Yaskawa INFORM job: A_ROOF_UPPER_0614_2_PAINT_29.JBI

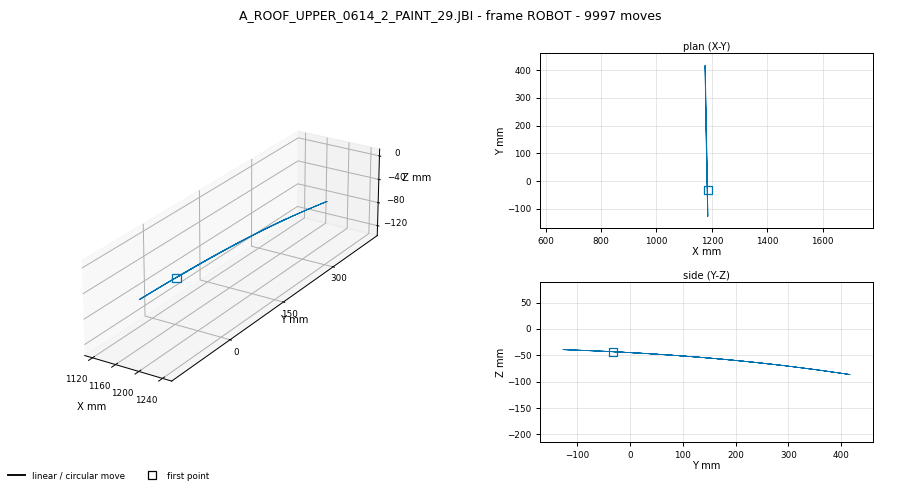
[picture p0: tool path of A_ROOF_UPPER_0614_2_PAINT_29.JBI in frame ROBOT, 9997 of 9997 moves have a stored position in this frame; points joined in program order, loops and branches not executed]
/JOB
//NAME A_ROOF_UPPER_0614_2_PAINT29
//POS
///NPOS 9997,0,0,0,0,0
///TOOL 1
///USER 0
///POSTYPE ROBOT
///RECTAN
///RCONF 1,0,0,0,0,0,0,0,0,0,0,0,0,0,0,0,0,0,0,0,0,0,0,0
C00000=1184.882,-32.072,-43.136,179.748,5.725,149.090
C00001=1184.877,-31.822,-43.149,179.750,5.725,149.089
C00002=1184.871,-31.573,-43.161,179.753,5.726,149.088
C00003=1184.866,-31.323,-43.173,179.755,5.726,149.088
C00004=1184.861,-31.074,-43.186,179.758,5.727,149.087
C00005=1184.855,-30.824,-43.198,179.760,5.727,149.086
C00006=1184.850,-30.574,-43.210,179.762,5.727,149.086
C00007=1184.846,-30.324,-43.223,179.765,5.728,149.085
C00008=1184.840,-30.074,-43.235,179.767,5.728,149.084
C00009=1184.835,-29.825,-43.248,179.770,5.729,149.084
C00010=1184.830,-29.576,-43.260,179.772,5.729,149.083
C00011=1184.825,-29.326,-43.272,179.775,5.730,149.083
C00012=1184.820,-29.077,-43.285,179.777,5.730,149.082
C00013=1184.815,-28.827,-43.298,179.780,5.730,149.081
C00014=1184.810,-28.577,-43.311,179.782,5.731,149.081
C00015=1184.804,-28.327,-43.322,179.784,5.731,149.080
C00016=1184.799,-28.078,-43.335,179.787,5.732,149.079
C00017=1184.794,-27.829,-43.348,179.789,5.733,149.079
C00018=1184.789,-27.579,-43.360,179.791,5.732,149.078
C00019=1184.784,-27.329,-43.372,179.794,5.733,149.077
C00020=1184.779,-27.079,-43.385,179.797,5.733,149.077
C00021=1184.773,-26.830,-43.398,179.799,5.734,149.076
C00022=1184.768,-26.580,-43.411,179.801,5.734,149.076
C00023=1184.763,-26.331,-43.423,179.804,5.735,149.075
C00024=1184.758,-26.081,-43.436,179.806,5.735,149.074
C00025=1184.753,-25.831,-43.448,179.808,5.735,149.074
C00026=1184.748,-25.582,-43.461,179.811,5.736,149.073
C00027=1184.743,-25.333,-43.474,179.814,5.736,149.072
C00028=1184.738,-25.083,-43.486,179.816,5.737,149.072
C00029=1184.732,-24.832,-43.499,179.819,5.738,149.071
C00030=1184.727,-24.583,-43.512,179.821,5.737,149.070
C00031=1184.722,-24.334,-43.524,179.823,5.738,149.070
C00032=1184.717,-24.084,-43.537,179.825,5.738,149.069
C00033=1184.712,-23.815,-43.550,179.828,5.739,149.069
C00034=1184.706,-23.545,-43.565,179.831,5.739,149.068
C00035=1184.701,-23.275,-43.578,179.833,5.740,149.067
C00036=1184.694,-23.005,-43.592,179.836,5.740,149.066
C00037=1184.689,-22.756,-43.604,179.839,5.741,149.066
C00038=1184.685,-22.506,-43.617,179.841,5.741,149.065
C00039=1184.680,-22.256,-43.630,179.844,5.742,149.065
C00040=1184.674,-22.007,-43.642,179.846,5.742,149.064
C00041=1184.669,-21.757,-43.656,179.848,5.742,149.063
C00042=1184.664,-21.507,-43.669,179.851,5.743,149.063
C00043=1184.659,-21.258,-43.681,179.853,5.743,149.062
C00044=1184.654,-21.009,-43.694,179.856,5.744,149.061
C00045=1184.649,-20.758,-43.707,179.858,5.744,149.061
C00046=1184.643,-20.509,-43.720,179.861,5.745,149.060
C00047=1184.638,-20.260,-43.732,179.863,5.745,149.060
C00048=1184.634,-20.010,-43.745,179.865,5.745,149.059
C00049=1184.628,-19.760,-43.759,179.868,5.746,149.058
C00050=1184.623,-19.511,-43.771,179.870,5.747,149.058
C00051=1184.618,-19.261,-43.784,179.873,5.747,149.057
C00052=1184.612,-19.011,-43.797,179.876,5.747,149.056
C00053=1184.607,-18.762,-43.810,179.878,5.748,149.056
C00054=1184.602,-18.512,-43.823,179.880,5.749,149.055
C00055=1184.598,-18.262,-43.836,179.882,5.748,149.054
C00056=1184.592,-18.013,-43.849,179.885,5.749,149.054
C00057=1184.587,-17.763,-43.861,179.887,5.750,149.053
C00058=1184.582,-17.513,-43.874,179.890,5.750,149.053
C00059=1184.576,-17.264,-43.888,179.893,5.751,149.052
C00060=1184.571,-17.015,-43.900,179.895,5.751,149.051
C00061=1184.567,-16.764,-43.913,179.897,5.752,149.051
C00062=1184.561,-16.515,-43.926,179.900,5.752,149.050
C00063=1184.556,-16.266,-43.940,179.902,5.752,149.049
C00064=1184.551,-16.016,-43.953,179.905,5.753,149.049
C00065=1184.546,-15.767,-43.966,179.907,5.753,149.048
C00066=1184.541,-15.516,-43.979,179.910,5.754,149.047
C00067=1184.536,-15.267,-43.991,179.912,5.754,149.047
C00068=1184.530,-15.018,-44.005,179.915,5.755,149.046
C00069=1184.526,-14.768,-44.018,179.917,5.756,149.046
C00070=1184.520,-14.518,-44.030,179.920,5.756,149.045
C00071=1184.515,-14.269,-44.044,179.922,5.757,149.044
C00072=1184.510,-14.019,-44.057,179.924,5.757,149.044
C00073=1184.505,-13.770,-44.070,179.927,5.757,149.043
C00074=1184.500,-13.520,-44.083,179.929,5.757,149.042
C00075=1184.495,-13.270,-44.096,179.932,5.758,149.042
C00076=1184.489,-13.021,-44.110,179.934,5.759,149.041
C00077=1184.485,-12.771,-44.123,179.937,5.759,149.041
C00078=1184.479,-12.522,-44.136,179.940,5.760,149.040
C00079=1184.474,-12.272,-44.149,179.942,5.761,149.039
C00080=1184.469,-12.023,-44.163,179.944,5.761,149.039
C00081=1184.464,-11.773,-44.176,179.947,5.761,149.038
C00082=1184.459,-11.523,-44.188,179.949,5.761,149.037
C00083=1184.453,-11.274,-44.201,179.951,5.762,149.037
C00084=1184.449,-11.024,-44.215,179.954,5.762,149.036
C00085=1184.443,-10.775,-44.228,179.957,5.763,149.035
C00086=1184.439,-10.525,-44.241,179.959,5.763,149.035
C00087=1184.433,-10.275,-44.255,179.961,5.764,149.034
C00088=1184.429,-10.025,-44.268,179.964,5.765,149.034
C00089=1184.423,-9.776,-44.281,179.967,5.765,149.033
C00090=1184.418,-9.526,-44.294,179.969,5.766,149.032
C00091=1184.413,-9.277,-44.308,179.972,5.766,149.032
C00092=1184.408,-9.027,-44.321,179.974,5.767,149.031
C00093=1184.402,-8.777,-44.334,179.976,5.767,149.030
C00094=1184.398,-8.528,-44.348,179.978,5.767,149.030
C00095=1184.392,-8.278,-44.361,179.981,5.768,149.029
C00096=1184.387,-8.029,-44.374,179.984,5.768,149.029
C00097=1184.382,-7.779,-44.388,179.986,5.769,149.028
C00098=1184.377,-7.530,-44.401,179.989,5.770,149.027
C00099=1184.372,-7.280,-44.415,179.991,5.770,149.027
C00100=1184.367,-7.031,-44.428,179.994,5.771,149.026
C00101=1184.362,-6.780,-44.441,179.996,5.771,149.026
C00102=1184.357,-6.532,-44.455,179.999,5.772,149.025
C00103=1184.352,-6.281,-44.468,-179.999,5.772,149.024
C00104=1184.346,-6.032,-44.482,-179.996,5.773,149.023
C00105=1184.342,-5.782,-44.495,-179.994,5.774,149.023
C00106=1184.337,-5.533,-44.509,-179.992,5.773,149.022
C00107=1184.331,-5.283,-44.522,-179.989,5.774,149.022
C00108=1184.327,-5.034,-44.536,-179.987,5.775,149.021
C00109=1184.321,-4.784,-44.549,-179.984,5.775,149.020
C00110=1184.316,-4.534,-44.562,-179.982,5.776,149.020
C00111=1184.311,-4.285,-44.576,-179.979,5.776,149.019
C00112=1184.306,-4.035,-44.589,-179.977,5.777,149.019
C00113=1184.301,-3.786,-44.603,-179.974,5.777,149.018
C00114=1184.295,-3.536,-44.617,-179.971,5.778,149.017
C00115=1184.290,-3.287,-44.630,-179.969,5.778,149.017
C00116=1184.285,-3.037,-44.644,-179.967,5.779,149.016
C00117=1184.280,-2.788,-44.657,-179.964,5.780,149.015
C00118=1184.275,-2.538,-44.671,-179.961,5.780,149.015
C00119=1184.270,-2.288,-44.685,-179.959,5.781,149.014
C00120=1184.265,-2.039,-44.698,-179.957,5.781,149.014
C00121=1184.260,-1.789,-44.712,-179.954,5.782,149.013
C00122=1184.255,-1.540,-44.725,-179.951,5.782,149.012
C00123=1184.250,-1.290,-44.738,-179.949,5.783,149.012
C00124=1184.245,-1.040,-44.753,-179.947,5.783,149.011
C00125=1184.239,-0.791,-44.767,-179.944,5.783,149.010
C00126=1184.234,-0.541,-44.780,-179.942,5.784,149.010
C00127=1184.229,-0.292,-44.794,-179.939,5.785,149.009
C00128=1184.224,-0.042,-44.808,-179.937,5.785,149.008
C00129=1184.219,0.208,-44.821,-179.934,5.786,149.008
C00130=1184.214,0.457,-44.835,-179.932,5.787,149.007
C00131=1184.209,0.707,-44.848,-179.929,5.787,149.007
C00132=1184.204,0.956,-44.862,-179.927,5.787,149.006
C00133=1184.199,1.206,-44.876,-179.925,5.788,149.006
C00134=1184.194,1.456,-44.889,-179.922,5.789,149.005
C00135=1184.189,1.705,-44.903,-179.919,5.789,149.004
C00136=1184.184,1.954,-44.918,-179.917,5.790,149.003
C00137=1184.178,2.224,-44.933,-179.914,5.790,149.003
C00138=1184.172,2.493,-44.947,-179.912,5.791,149.002
C00139=1184.167,2.762,-44.962,-179.909,5.792,149.002
C00140=1184.162,3.031,-44.977,-179.906,5.793,149.001
C00141=1184.157,3.281,-44.991,-179.903,5.793,149.000
C00142=1184.151,3.530,-45.005,-179.901,5.794,149.000
C00143=1184.146,3.780,-45.018,-179.898,5.795,148.999
C00144=1184.141,4.030,-45.033,-179.896,5.795,148.998
C00145=1184.136,4.279,-45.046,-179.894,5.795,148.998
C00146=1184.131,4.528,-45.060,-179.891,5.795,148.997
C00147=1184.126,4.779,-45.074,-179.889,5.796,148.997
C00148=1184.121,5.028,-45.088,-179.886,5.797,148.996
C00149=1184.116,5.277,-45.102,-179.884,5.797,148.995
C00150=1184.111,5.527,-45.116,-179.881,5.798,148.995
C00151=1184.106,5.776,-45.130,-179.879,5.798,148.994
C00152=1184.101,6.026,-45.143,-179.876,5.799,148.993
C00153=1184.096,6.276,-45.157,-179.873,5.799,148.993
C00154=1184.091,6.525,-45.172,-179.871,5.800,148.992
C00155=1184.085,6.774,-45.186,-179.869,5.801,148.992
C00156=1184.080,7.024,-45.200,-179.866,5.801,148.991
C00157=1184.075,7.274,-45.214,-179.864,5.802,148.990
C00158=1184.070,7.523,-45.227,-179.861,5.802,148.990
C00159=1184.065,7.773,-45.241,-179.858,5.803,148.989
C00160=1184.060,8.023,-45.255,-179.856,5.803,148.988
C00161=1184.055,8.272,-45.270,-179.854,5.804,148.988
C00162=1184.050,8.521,-45.283,-179.851,5.805,148.987
C00163=1184.045,8.771,-45.298,-179.848,5.805,148.986
C00164=1184.040,9.021,-45.312,-179.846,5.806,148.986
C00165=1184.035,9.270,-45.326,-179.844,5.807,148.985
C00166=1184.029,9.519,-45.340,-179.841,5.807,148.985
C00167=1184.024,9.769,-45.354,-179.839,5.808,148.984
C00168=1184.019,10.019,-45.369,-179.836,5.808,148.984
C00169=1184.014,10.269,-45.383,-179.833,5.809,148.983
C00170=1184.009,10.518,-45.397,-179.831,5.809,148.982
C00171=1184.004,10.767,-45.411,-179.828,5.811,148.982
C00172=1184.000,11.017,-45.425,-179.825,5.812,148.981
C00173=1183.995,11.266,-45.439,-179.823,5.812,148.980
C00174=1183.989,11.515,-45.453,-179.821,5.813,148.980
C00175=1183.984,11.765,-45.467,-179.818,5.813,148.979
C00176=1183.979,12.015,-45.482,-179.815,5.814,148.979
C00177=1183.974,12.265,-45.496,-179.813,5.815,148.978
C00178=1183.969,12.514,-45.510,-179.810,5.815,148.977
C00179=1183.964,12.763,-45.524,-179.808,5.816,148.977
C00180=1183.959,13.013,-45.538,-179.805,5.816,148.976
C00181=1183.954,13.263,-45.553,-179.803,5.817,148.976
C00182=1183.949,13.512,-45.567,-179.800,5.817,148.975
C00183=1183.943,13.762,-45.582,-179.798,5.818,148.974
C00184=1183.938,14.011,-45.596,-179.795,5.819,148.974
C00185=1183.933,14.261,-45.610,-179.793,5.819,148.973
C00186=1183.928,14.511,-45.624,-179.790,5.820,148.972
C00187=1183.923,14.760,-45.639,-179.788,5.821,148.972
C00188=1183.918,15.010,-45.654,-179.785,5.821,148.971
C00189=1183.913,15.259,-45.668,-179.783,5.822,148.971
C00190=1183.908,15.508,-45.682,-179.780,5.822,148.970
C00191=1183.903,15.758,-45.696,-179.778,5.823,148.969
C00192=1183.898,16.008,-45.710,-179.775,5.823,148.969
C00193=1183.893,16.257,-45.725,-179.773,5.824,148.968
C00194=1183.888,16.507,-45.740,-179.770,5.825,148.968
C00195=1183.883,16.756,-45.754,-179.768,5.825,148.967
C00196=1183.878,17.006,-45.768,-179.765,5.826,148.966
C00197=1183.873,17.256,-45.783,-179.763,5.827,148.966
C00198=1183.867,17.505,-45.797,-179.760,5.827,148.965
C00199=1183.862,17.754,-45.812,-179.757,5.828,148.964
C00200=1183.857,18.004,-45.826,-179.754,5.829,148.964
C00201=1183.852,18.254,-45.840,-179.752,5.830,148.963
C00202=1183.848,18.503,-45.855,-179.750,5.830,148.963
C00203=1183.843,18.752,-45.870,-179.747,5.831,148.962
C00204=1183.837,19.002,-45.885,-179.745,5.832,148.961
C00205=1183.832,19.252,-45.899,-179.742,5.832,148.961
C00206=1183.827,19.502,-45.913,-179.740,5.833,148.960
C00207=1183.822,19.750,-45.928,-179.737,5.833,148.960
C00208=1183.817,20.000,-45.942,-179.735,5.834,148.959
C00209=1183.812,20.250,-45.956,-179.732,5.834,148.958
C00210=1183.807,20.499,-45.972,-179.730,5.835,148.958
C00211=1183.802,20.749,-45.986,-179.727,5.836,148.957
C00212=1183.797,20.998,-46.000,-179.725,5.836,148.956
C00213=1183.792,21.248,-46.015,-179.722,5.837,148.956
C00214=1183.787,21.497,-46.030,-179.720,5.838,148.955
C00215=1183.782,21.747,-46.045,-179.717,5.839,148.955
C00216=1183.777,21.996,-46.060,-179.714,5.840,148.954
C00217=1183.772,22.246,-46.074,-179.712,5.840,148.953
C00218=1183.767,22.495,-46.089,-179.709,5.841,148.953
C00219=1183.762,22.745,-46.104,-179.706,5.841,148.952
C00220=1183.757,22.995,-46.118,-179.704,5.842,148.952
C00221=1183.752,23.244,-46.133,-179.702,5.843,148.951
C00222=1183.747,23.494,-46.147,-179.699,5.843,148.950
C00223=1183.742,23.743,-46.163,-179.697,5.844,148.950
C00224=1183.737,23.993,-46.177,-179.694,5.844,148.949
C00225=1183.732,24.243,-46.191,-179.692,5.845,148.948
C00226=1183.727,24.492,-46.206,-179.689,5.846,148.948
C00227=1183.721,24.742,-46.221,-179.686,5.847,148.947
C00228=1183.717,24.991,-46.236,-179.684,5.848,148.947
C00229=1183.712,25.240,-46.251,-179.681,5.848,148.946
C00230=1183.706,25.490,-46.266,-179.679,5.849,148.946
C00231=1183.701,25.740,-46.280,-179.676,5.849,148.945
C00232=1183.697,25.989,-46.295,-179.674,5.850,148.944
C00233=1183.691,26.239,-46.310,-179.671,5.851,148.944
C00234=1183.686,26.488,-46.325,-179.669,5.851,148.943
C00235=1183.681,26.738,-46.340,-179.666,5.852,148.943
C00236=1183.676,26.987,-46.355,-179.664,5.853,148.942
C00237=1183.671,27.237,-46.369,-179.661,5.854,148.941
C00238=1183.666,27.486,-46.384,-179.658,5.855,148.941
C00239=1183.661,27.735,-46.400,-179.656,5.855,148.940
C00240=1183.656,27.985,-46.414,-179.653,5.856,148.939
C00241=1183.650,28.254,-46.431,-179.650,5.856,148.939
C00242=1183.645,28.523,-46.446,-179.648,5.857,148.938
C00243=1183.640,28.791,-46.463,-179.645,5.858,148.938
C00244=1183.634,29.060,-46.479,-179.642,5.859,148.937
C00245=1183.630,29.310,-46.493,-179.640,5.859,148.936
C00246=1183.624,29.559,-46.509,-179.637,5.860,148.936
C00247=1183.619,29.808,-46.524,-179.635,5.861,148.935
C00248=1183.614,30.058,-46.539,-179.632,5.861,148.934
C00249=1183.609,30.307,-46.554,-179.629,5.863,148.934
C00250=1183.604,30.557,-46.569,-179.627,5.864,148.933
C00251=1183.599,30.806,-46.584,-179.624,5.864,148.933
C00252=1183.594,31.056,-46.599,-179.622,5.865,148.932
C00253=1183.589,31.305,-46.614,-179.620,5.865,148.932
C00254=1183.584,31.555,-46.629,-179.617,5.866,148.931
C00255=1183.579,31.805,-46.644,-179.614,5.866,148.930
C00256=1183.574,32.054,-46.659,-179.611,5.868,148.930
C00257=1183.569,32.303,-46.675,-179.609,5.869,148.929
C00258=1183.564,32.553,-46.689,-179.606,5.869,148.928
C00259=1183.559,32.802,-46.705,-179.604,5.870,148.928
C00260=1183.554,33.051,-46.720,-179.601,5.870,148.927
C00261=1183.548,33.301,-46.735,-179.599,5.871,148.927
C00262=1183.544,33.551,-46.750,-179.597,5.872,148.926
C00263=1183.539,33.801,-46.766,-179.594,5.872,148.925
C00264=1183.534,34.050,-46.781,-179.591,5.874,148.925
C00265=1183.529,34.299,-46.796,-179.589,5.874,148.924
C00266=1183.524,34.549,-46.811,-179.586,5.875,148.924
C00267=1183.518,34.798,-46.826,-179.584,5.876,148.923
C00268=1183.514,35.047,-46.841,-179.581,5.876,148.923
C00269=1183.509,35.297,-46.857,-179.578,5.877,148.922
C00270=1183.504,35.547,-46.872,-179.576,5.879,148.921
C00271=1183.499,35.796,-46.888,-179.573,5.879,148.921
C00272=1183.493,36.046,-46.903,-179.570,5.880,148.920
C00273=1183.489,36.295,-46.918,-179.568,5.880,148.920
C00274=1183.483,36.544,-46.933,-179.566,5.881,148.919
C00275=1183.479,36.794,-46.948,-179.563,5.881,148.918
C00276=1183.474,37.044,-46.964,-179.561,5.882,148.918
C00277=1183.468,37.293,-46.980,-179.558,5.884,148.917
C00278=1183.464,37.542,-46.995,-179.555,5.884,148.916
C00279=1183.458,37.792,-47.010,-179.553,5.885,148.916
C00280=1183.454,38.042,-47.025,-179.550,5.886,148.915
C00281=1183.449,38.291,-47.040,-179.548,5.886,148.915
C00282=1183.443,38.541,-47.056,-179.545,5.887,148.914
C00283=1183.439,38.790,-47.071,-179.542,5.888,148.914
C00284=1183.433,39.039,-47.087,-179.540,5.889,148.913
C00285=1183.428,39.289,-47.103,-179.537,5.890,148.912
C00286=1183.424,39.538,-47.118,-179.535,5.890,148.912
C00287=1183.418,39.788,-47.133,-179.533,5.891,148.911
C00288=1183.413,40.037,-47.149,-179.530,5.891,148.911
C00289=1183.409,40.287,-47.164,-179.527,5.893,148.910
C00290=1183.404,40.536,-47.180,-179.525,5.894,148.910
C00291=1183.398,40.786,-47.195,-179.522,5.894,148.909
C00292=1183.394,41.035,-47.210,-179.519,5.895,148.908
C00293=1183.389,41.285,-47.226,-179.517,5.896,148.908
C00294=1183.383,41.534,-47.242,-179.514,5.897,148.907
C00295=1183.378,41.784,-47.257,-179.511,5.897,148.906
C00296=1183.373,42.033,-47.272,-179.509,5.898,148.906
C00297=1183.369,42.283,-47.288,-179.506,5.899,148.905
C00298=1183.364,42.532,-47.305,-179.504,5.900,148.905
C00299=1183.359,42.781,-47.320,-179.501,5.901,148.904
C00300=1183.353,43.030,-47.335,-179.498,5.901,148.904
C00301=1183.349,43.280,-47.351,-179.496,5.902,148.903
C00302=1183.343,43.530,-47.367,-179.494,5.903,148.902
C00303=1183.339,43.779,-47.382,-179.491,5.903,148.902
C00304=1183.334,44.029,-47.398,-179.488,5.905,148.901
C00305=1183.328,44.278,-47.413,-179.486,5.906,148.901
C00306=1183.323,44.527,-47.430,-179.483,5.906,148.900
C00307=1183.319,44.777,-47.446,-179.481,5.907,148.899
C00308=1183.314,45.026,-47.461,-179.478,5.907,148.899
C00309=1183.309,45.276,-47.476,-179.475,5.909,148.898
C00310=1183.304,45.526,-47.492,-179.473,5.910,148.898
C00311=1183.298,45.775,-47.508,-179.470,5.910,148.897
C00312=1183.293,46.024,-47.524,-179.468,5.911,148.897
C00313=1183.289,46.274,-47.539,-179.465,5.912,148.896
C00314=1183.284,46.523,-47.555,-179.463,5.913,148.895
C00315=1183.279,46.773,-47.571,-179.460,5.914,148.895
C00316=1183.274,47.022,-47.587,-179.457,5.914,148.894
C00317=1183.269,47.272,-47.603,-179.455,5.915,148.894
C00318=1183.263,47.521,-47.618,-179.453,5.916,148.893
C00319=1183.259,47.771,-47.634,-179.449,5.917,148.892
C00320=1183.254,48.020,-47.650,-179.447,5.918,148.892
C00321=1183.249,48.269,-47.666,-179.445,5.918,148.891
C00322=1183.244,48.519,-47.682,-179.442,5.919,148.891
C00323=1183.239,48.768,-47.697,-179.439,5.921,148.890
C00324=1183.234,49.018,-47.714,-179.437,5.921,148.889
C00325=1183.229,49.267,-47.729,-179.434,5.922,148.889
C00326=1183.223,49.517,-47.745,-179.432,5.922,148.888
C00327=1183.219,49.766,-47.762,-179.429,5.924,148.888
C00328=1183.214,50.015,-47.777,-179.426,5.925,148.887
C00329=1183.210,50.265,-47.793,-179.424,5.925,148.887
C00330=1183.204,50.514,-47.809,-179.422,5.926,148.886
C00331=1183.199,50.764,-47.825,-179.419,5.927,148.885
C00332=1183.194,51.013,-47.841,-179.416,5.928,148.885
C00333=1183.189,51.262,-47.857,-179.414,5.929,148.884
C00334=1183.184,51.513,-47.873,-179.411,5.929,148.884
C00335=1183.179,51.761,-47.889,-179.409,5.930,148.883
C00336=1183.174,52.011,-47.905,-179.406,5.932,148.883
C00337=1183.169,52.260,-47.921,-179.403,5.932,148.882
C00338=1183.165,52.510,-47.937,-179.401,5.933,148.881
C00339=1183.159,52.759,-47.954,-179.398,5.933,148.881
C00340=1183.154,53.009,-47.969,-179.395,5.935,148.880
C00341=1183.150,53.258,-47.986,-179.393,5.936,148.880
C00342=1183.144,53.507,-48.001,-179.390,5.936,148.879
C00343=1183.139,53.758,-48.017,-179.388,5.937,148.879
C00344=1183.134,54.006,-48.034,-179.385,5.938,148.878
C00345=1183.129,54.276,-48.051,-179.382,5.939,148.877
C00346=1183.124,54.543,-48.069,-179.379,5.941,148.877
C00347=1183.119,54.812,-48.086,-179.377,5.941,148.876
C00348=1183.113,55.080,-48.103,-179.374,5.942,148.876
C00349=1183.109,55.330,-48.119,-179.371,5.943,148.875
C00350=1183.103,55.579,-48.135,-179.369,5.944,148.874
C00351=1183.099,55.829,-48.152,-179.366,5.944,148.874
C00352=1183.093,56.078,-48.168,-179.363,5.946,148.873
C00353=1183.088,56.328,-48.185,-179.361,5.947,148.873
C00354=1183.083,56.577,-48.201,-179.359,5.947,148.872
C00355=1183.078,56.827,-48.217,-179.356,5.948,148.872
C00356=1183.073,57.076,-48.233,-179.353,5.949,148.871
C00357=1183.068,57.326,-48.249,-179.351,5.950,148.870
C00358=1183.063,57.574,-48.265,-179.348,5.951,148.870
C00359=1183.059,57.824,-48.282,-179.346,5.952,148.869
C00360=1183.054,58.074,-48.298,-179.343,5.953,148.869
C00361=1183.049,58.323,-48.314,-179.340,5.953,148.868
C00362=1183.044,58.573,-48.332,-179.338,5.954,148.868
C00363=1183.038,58.822,-48.347,-179.335,5.956,148.867
C00364=1183.034,59.072,-48.364,-179.332,5.957,148.866
C00365=1183.029,59.320,-48.380,-179.330,5.957,148.866
C00366=1183.024,59.570,-48.396,-179.328,5.958,148.865
C00367=1183.019,59.819,-48.412,-179.324,5.959,148.865
C00368=1183.014,60.069,-48.430,-179.322,5.960,148.864
C00369=1183.009,60.319,-48.446,-179.320,5.961,148.864
C00370=1183.004,60.568,-48.462,-179.316,5.962,148.863
C00371=1182.999,60.817,-48.479,-179.314,5.963,148.863
C00372=1182.994,61.066,-48.495,-179.312,5.963,148.862
C00373=1182.989,61.317,-48.511,-179.309,5.965,148.861
C00374=1182.984,61.565,-48.528,-179.306,5.966,148.861
C00375=1182.979,61.815,-48.544,-179.304,5.966,148.860
C00376=1182.975,62.064,-48.561,-179.302,5.967,148.860
C00377=1182.970,62.313,-48.577,-179.298,5.968,148.859
C00378=1182.964,62.564,-48.594,-179.296,5.969,148.859
C00379=1182.959,62.812,-48.610,-179.294,5.970,148.858
C00380=1182.954,63.062,-48.627,-179.291,5.972,148.857
C00381=1182.950,63.311,-48.644,-179.288,5.972,148.857
C00382=1182.944,63.560,-48.660,-179.286,5.973,148.856
C00383=1182.940,63.810,-48.677,-179.283,5.974,148.856
C00384=1182.935,64.060,-48.693,-179.280,5.975,148.855
C00385=1182.930,64.309,-48.709,-179.278,5.976,148.855
C00386=1182.925,64.559,-48.727,-179.275,5.977,148.854
C00387=1182.920,64.808,-48.743,-179.273,5.978,148.854
C00388=1182.915,65.057,-48.760,-179.270,5.978,148.853
C00389=1182.910,65.307,-48.777,-179.267,5.980,148.852
C00390=1182.905,65.556,-48.794,-179.265,5.981,148.852
C00391=1182.900,65.805,-48.810,-179.262,5.981,148.851
C00392=1182.895,66.055,-48.827,-179.259,5.983,148.851
C00393=1182.891,66.304,-48.844,-179.257,5.983,148.850
C00394=1182.886,66.553,-48.860,-179.255,5.984,148.850
C00395=1182.880,66.803,-48.877,-179.251,5.986,148.849
C00396=1182.876,67.053,-48.893,-179.249,5.987,148.848
C00397=1182.870,67.302,-48.910,-179.247,5.987,148.848
C00398=1182.865,67.551,-48.927,-179.244,5.989,148.847
C00399=1182.861,67.801,-48.944,-179.241,5.989,148.847
C00400=1182.856,68.050,-48.960,-179.239,5.990,148.846
C00401=1182.851,68.299,-48.978,-179.236,5.992,148.846
C00402=1182.846,68.548,-48.995,-179.233,5.992,148.845
C00403=1182.841,68.798,-49.012,-179.231,5.993,148.845
C00404=1182.836,69.047,-49.028,-179.228,5.994,148.844
C00405=1182.831,69.296,-49.045,-179.226,5.995,148.843
C00406=1182.826,69.546,-49.062,-179.223,5.996,148.843
C00407=1182.822,69.796,-49.079,-179.220,5.997,148.842
C00408=1182.816,70.045,-49.096,-179.218,5.998,148.842
C00409=1182.811,70.294,-49.112,-179.216,5.999,148.841
C00410=1182.807,70.544,-49.129,-179.212,6.000,148.841
C00411=1182.801,70.793,-49.146,-179.210,6.001,148.840
C00412=1182.797,71.042,-49.162,-179.207,6.002,148.840
C00413=1182.791,71.292,-49.180,-179.204,6.003,148.839
C00414=1182.787,71.541,-49.197,-179.202,6.004,148.838
C00415=1182.782,71.791,-49.214,-179.199,6.005,148.838
C00416=1182.777,72.040,-49.231,-179.197,6.006,148.837
C00417=1182.772,72.289,-49.248,-179.194,6.007,148.837
C00418=1182.767,72.539,-49.265,-179.191,6.008,148.836
C00419=1182.762,72.789,-49.282,-179.189,6.009,148.836
C00420=1182.757,73.037,-49.299,-179.187,6.010,148.835
C00421=1182.752,73.287,-49.316,-179.184,6.011,148.835
C00422=1182.748,73.536,-49.333,-179.181,6.012,148.834
C00423=1182.742,73.786,-49.350,-179.178,6.013,148.833
C00424=1182.738,74.035,-49.368,-179.176,6.014,148.833
C00425=1182.732,74.284,-49.384,-179.173,6.015,148.832
C00426=1182.728,74.533,-49.401,-179.171,6.017,148.832
C00427=1182.723,74.783,-49.418,-179.168,6.017,148.831
C00428=1182.718,75.032,-49.436,-179.166,6.018,148.831
C00429=1182.713,75.282,-49.453,-179.163,6.019,148.830
C00430=1182.708,75.532,-49.470,-179.160,6.020,148.830
C00431=1182.703,75.780,-49.487,-179.157,6.022,148.829
C00432=1182.698,76.029,-49.505,-179.155,6.022,148.828
C00433=1182.694,76.279,-49.521,-179.153,6.023,148.828
C00434=1182.688,76.529,-49.538,-179.149,6.024,148.827
C00435=1182.683,76.778,-49.556,-179.147,6.025,148.827
C00436=1182.679,77.027,-49.573,-179.144,6.027,148.826
C00437=1182.673,77.277,-49.590,-179.142,6.027,148.826
C00438=1182.669,77.525,-49.607,-179.139,6.028,148.825
C00439=1182.664,77.775,-49.625,-179.137,6.030,148.825
C00440=1182.659,78.024,-49.643,-179.134,6.030,148.824
C00441=1182.654,78.274,-49.659,-179.131,6.032,148.824
C00442=1182.649,78.524,-49.677,-179.129,6.033,148.823
C00443=1182.644,78.773,-49.695,-179.126,6.033,148.823
C00444=1182.640,79.022,-49.711,-179.123,6.035,148.822
C00445=1182.634,79.271,-49.729,-179.121,6.036,148.822
C00446=1182.629,79.521,-49.746,-179.118,6.037,148.821
C00447=1182.625,79.769,-49.763,-179.116,6.038,148.820
C00448=1182.620,80.019,-49.781,-179.112,6.039,148.820
C00449=1182.614,80.288,-49.799,-179.110,6.040,148.819
C00450=1182.609,80.556,-49.819,-179.107,6.042,148.819
C00451=1182.604,80.824,-49.837,-179.105,6.042,148.818
C00452=1182.599,81.092,-49.856,-179.102,6.044,148.818
C00453=1182.594,81.342,-49.873,-179.099,6.044,148.817
C00454=1182.589,81.591,-49.891,-179.096,6.046,148.817
C00455=1182.584,81.841,-49.908,-179.094,6.047,148.816
C00456=1182.579,82.090,-49.926,-179.091,6.048,148.815
C00457=1182.574,82.340,-49.943,-179.088,6.049,148.815
C00458=1182.569,82.589,-49.961,-179.086,6.051,148.814
C00459=1182.564,82.839,-49.978,-179.083,6.051,148.814
C00460=1182.560,83.088,-49.996,-179.081,6.052,148.813
C00461=1182.555,83.338,-50.013,-179.078,6.053,148.813
C00462=1182.550,83.587,-50.031,-179.076,6.054,148.812
C00463=1182.545,83.836,-50.049,-179.072,6.056,148.812
C00464=1182.540,84.085,-50.066,-179.070,6.056,148.811
C00465=1182.535,84.335,-50.084,-179.067,6.058,148.811
C00466=1182.530,84.584,-50.102,-179.065,6.059,148.810
C00467=1182.525,84.834,-50.119,-179.062,6.059,148.809
C00468=1182.520,85.083,-50.137,-179.060,6.061,148.809
C00469=1182.515,85.332,-50.155,-179.057,6.062,148.808
C00470=1182.511,85.581,-50.172,-179.054,6.063,148.808
C00471=1182.506,85.831,-50.190,-179.052,6.064,148.808
C00472=1182.501,86.080,-50.207,-179.049,6.066,148.807
C00473=1182.496,86.329,-50.225,-179.047,6.066,148.806
C00474=1182.491,86.579,-50.243,-179.044,6.068,148.806
C00475=1182.486,86.828,-50.261,-179.041,6.069,148.805
C00476=1182.481,87.078,-50.278,-179.038,6.070,148.805
C00477=1182.477,87.326,-50.295,-179.036,6.071,148.804
C00478=1182.472,87.576,-50.313,-179.033,6.072,148.804
C00479=1182.467,87.825,-50.331,-179.031,6.073,148.803
C00480=1182.462,88.074,-50.349,-179.028,6.074,148.803
C00481=1182.457,88.324,-50.367,-179.025,6.075,148.802
C00482=1182.452,88.573,-50.385,-179.023,6.076,148.802
C00483=1182.447,88.822,-50.403,-179.020,6.078,148.801
C00484=1182.442,89.071,-50.421,-179.017,6.078,148.800
C00485=1182.437,89.321,-50.438,-179.015,6.080,148.800
C00486=1182.432,89.570,-50.456,-179.013,6.081,148.800
C00487=1182.427,89.819,-50.474,-179.009,6.082,148.799
C00488=1182.422,90.069,-50.492,-179.007,6.083,148.799
C00489=1182.417,90.318,-50.510,-179.004,6.085,148.798
C00490=1182.412,90.567,-50.528,-179.002,6.085,148.797
C00491=1182.409,90.817,-50.545,-178.999,6.087,148.797
C00492=1182.404,91.066,-50.563,-178.997,6.088,148.796
C00493=1182.399,91.316,-50.581,-178.993,6.089,148.796
C00494=1182.394,91.565,-50.599,-178.991,6.090,148.795
C00495=1182.389,91.814,-50.617,-178.989,6.092,148.795
C00496=1182.384,92.063,-50.635,-178.986,6.092,148.794
C00497=1182.379,92.312,-50.653,-178.983,6.094,148.794
C00498=1182.373,92.562,-50.671,-178.981,6.095,148.793
C00499=1182.368,92.811,-50.689,-178.978,6.096,148.793
C00500=1182.364,93.061,-50.707,-178.975,6.097,148.792
C00501=1182.359,93.310,-50.725,-178.972,6.099,148.792
C00502=1182.354,93.559,-50.743,-178.970,6.099,148.791
C00503=1182.349,93.808,-50.761,-178.967,6.101,148.791
C00504=1182.344,94.057,-50.779,-178.965,6.102,148.790
C00505=1182.339,94.307,-50.797,-178.962,6.103,148.790
C00506=1182.335,94.556,-50.815,-178.960,6.104,148.789
C00507=1182.330,94.806,-50.834,-178.956,6.105,148.789
C00508=1182.325,95.055,-50.852,-178.954,6.106,148.788
C00509=1182.320,95.304,-50.870,-178.951,6.108,148.788
C00510=1182.315,95.553,-50.888,-178.949,6.109,148.787
C00511=1182.311,95.802,-50.906,-178.946,6.110,148.787
C00512=1182.306,96.053,-50.925,-178.944,6.111,148.786
C00513=1182.301,96.302,-50.943,-178.941,6.113,148.786
C00514=1182.296,96.550,-50.961,-178.938,6.113,148.785
C00515=1182.291,96.800,-50.979,-178.936,6.115,148.785
C00516=1182.286,97.049,-50.997,-178.933,6.116,148.784
C00517=1182.282,97.299,-51.016,-178.930,6.117,148.783
C00518=1182.277,97.548,-51.034,-178.928,6.118,148.783
C00519=1182.271,97.797,-51.052,-178.925,6.119,148.782
C00520=1182.266,98.046,-51.070,-178.923,6.120,148.782
C00521=1182.262,98.295,-51.089,-178.920,6.122,148.781
C00522=1182.257,98.545,-51.107,-178.917,6.123,148.781
C00523=1182.253,98.794,-51.125,-178.915,6.124,148.781
C00524=1182.247,99.044,-51.144,-178.912,6.126,148.780
C00525=1182.242,99.293,-51.162,-178.909,6.127,148.779
C00526=1182.238,99.542,-51.181,-178.906,6.128,148.779
C00527=1182.233,99.791,-51.199,-178.904,6.129,148.778
C00528=1182.228,100.040,-51.217,-178.901,6.131,148.778
C00529=1182.223,100.290,-51.235,-178.899,6.131,148.777
C00530=1182.218,100.540,-51.254,-178.896,6.133,148.777
C00531=1182.214,100.788,-51.272,-178.893,6.133,148.776
C00532=1182.209,101.037,-51.290,-178.891,6.135,148.776
C00533=1182.203,101.287,-51.309,-178.889,6.136,148.775
C00534=1182.199,101.536,-51.328,-178.885,6.137,148.775
C00535=1182.194,101.785,-51.346,-178.883,6.139,148.774
C00536=1182.189,102.034,-51.364,-178.880,6.140,148.774
C00537=1182.184,102.284,-51.384,-178.877,6.141,148.773
C00538=1182.180,102.533,-51.402,-178.875,6.142,148.773
C00539=1182.175,102.782,-51.419,-178.872,6.144,148.772
C00540=1182.169,103.031,-51.439,-178.870,6.145,148.772
C00541=1182.165,103.281,-51.457,-178.867,6.146,148.771
C00542=1182.160,103.530,-51.475,-178.864,6.148,148.771
C00543=1182.155,103.779,-51.494,-178.862,6.149,148.770
C00544=1182.150,104.029,-51.513,-178.859,6.150,148.770
C00545=1182.146,104.278,-51.531,-178.857,6.151,148.769
C00546=1182.140,104.527,-51.550,-178.854,6.153,148.769
C00547=1182.136,104.777,-51.568,-178.851,6.153,148.768
C00548=1182.131,105.026,-51.587,-178.849,6.155,148.768
C00549=1182.126,105.275,-51.606,-178.845,6.156,148.767
C00550=1182.122,105.524,-51.625,-178.843,6.157,148.767
C00551=1182.116,105.774,-51.643,-178.840,6.159,148.766
C00552=1182.112,106.023,-51.662,-178.838,6.160,148.766
C00553=1182.106,106.292,-51.682,-178.835,6.161,148.765
C00554=1182.101,106.560,-51.702,-178.832,6.163,148.765
C00555=1182.096,106.828,-51.722,-178.829,6.164,148.764
C00556=1182.091,107.097,-51.742,-178.827,6.165,148.764
C00557=1182.086,107.346,-51.762,-178.824,6.167,148.763
C00558=1182.081,107.595,-51.780,-178.821,6.168,148.763
C00559=1182.076,107.844,-51.799,-178.819,6.169,148.762
C00560=1182.071,108.093,-51.818,-178.816,6.171,148.762
C00561=1182.067,108.343,-51.836,-178.813,6.171,148.761
C00562=1182.062,108.592,-51.855,-178.811,6.173,148.761
C00563=1182.057,108.842,-51.874,-178.808,6.175,148.760
C00564=1182.052,109.090,-51.893,-178.805,6.175,148.760
C00565=1182.047,109.340,-51.911,-178.803,6.177,148.759
C00566=1182.042,109.589,-51.931,-178.800,6.178,148.759
C00567=1182.038,109.838,-51.949,-178.797,6.179,148.758
C00568=1182.033,110.088,-51.968,-178.794,6.181,148.758
C00569=1182.028,110.336,-51.987,-178.792,6.182,148.758
C00570=1182.023,110.586,-52.007,-178.789,6.183,148.757
C00571=1182.019,110.835,-52.025,-178.787,6.184,148.756
C00572=1182.013,111.084,-52.044,-178.784,6.186,148.756
C00573=1182.009,111.333,-52.063,-178.781,6.187,148.755
C00574=1182.004,111.583,-52.082,-178.779,6.188,148.755
C00575=1181.999,111.832,-52.101,-178.776,6.190,148.754
C00576=1181.994,112.081,-52.120,-178.773,6.191,148.754
C00577=1181.989,112.330,-52.140,-178.771,6.192,148.754
C00578=1181.985,112.580,-52.158,-178.768,6.194,148.753
C00579=1181.980,112.829,-52.177,-178.766,6.195,148.753
C00580=1181.975,113.078,-52.196,-178.763,6.196,148.752
C00581=1181.970,113.327,-52.216,-178.760,6.198,148.752
C00582=1181.965,113.577,-52.234,-178.758,6.199,148.751
C00583=1181.961,113.826,-52.253,-178.755,6.200,148.751
C00584=1181.955,114.075,-52.273,-178.752,6.202,148.750
C00585=1181.951,114.325,-52.292,-178.750,6.203,148.750
C00586=1181.946,114.573,-52.311,-178.747,6.204,148.749
C00587=1181.941,114.823,-52.330,-178.744,6.206,148.749
C00588=1181.936,115.072,-52.349,-178.742,6.207,148.748
C00589=1181.932,115.321,-52.368,-178.739,6.208,148.748
C00590=1181.926,115.570,-52.388,-178.737,6.209,148.747
C00591=1181.922,115.820,-52.407,-178.734,6.211,148.747
C00592=1181.917,116.068,-52.426,-178.731,6.213,148.746
C00593=1181.912,116.318,-52.446,-178.729,6.213,148.746
C00594=1181.908,116.567,-52.464,-178.726,6.215,148.745
C00595=1181.903,116.817,-52.483,-178.723,6.217,148.745
C00596=1181.897,117.066,-52.502,-178.721,6.218,148.745
C00597=1181.893,117.315,-52.522,-178.718,6.219,148.744
C00598=1181.889,117.564,-52.541,-178.715,6.221,148.744
C00599=1181.883,117.813,-52.560,-178.713,6.222,148.743
C00600=1181.878,118.063,-52.580,-178.710,6.223,148.742
C00601=1181.874,118.311,-52.599,-178.707,6.225,148.742
C00602=1181.869,118.561,-52.618,-178.705,6.226,148.742
C00603=1181.864,118.810,-52.638,-178.701,6.227,148.741
C00604=1181.859,119.059,-52.657,-178.699,6.229,148.741
C00605=1181.855,119.309,-52.676,-178.697,6.230,148.740
C00606=1181.850,119.558,-52.696,-178.694,6.231,148.740
C00607=1181.845,119.807,-52.715,-178.691,6.233,148.739
C00608=1181.840,120.057,-52.735,-178.689,6.234,148.739
C00609=1181.835,120.306,-52.754,-178.686,6.235,148.738
C00610=1181.831,120.555,-52.773,-178.683,6.237,148.738
C00611=1181.825,120.804,-52.793,-178.681,6.238,148.737
C00612=1181.821,121.053,-52.813,-178.678,6.240,148.737
C00613=1181.816,121.302,-52.833,-178.675,6.241,148.737
C00614=1181.811,121.551,-52.852,-178.673,6.242,148.736
C00615=1181.807,121.800,-52.871,-178.670,6.244,148.736
C00616=1181.802,122.050,-52.891,-178.667,6.245,148.735
C00617=1181.797,122.299,-52.910,-178.664,6.247,148.735
C00618=1181.792,122.548,-52.930,-178.662,6.248,148.734
C00619=1181.787,122.798,-52.949,-178.659,6.249,148.734
C00620=1181.782,123.046,-52.969,-178.656,6.251,148.733
C00621=1181.778,123.296,-52.989,-178.654,6.252,148.733
C00622=1181.774,123.545,-53.008,-178.651,6.253,148.732
C00623=1181.768,123.794,-53.027,-178.648,6.255,148.732
C00624=1181.764,124.043,-53.047,-178.646,6.256,148.731
C00625=1181.759,124.292,-53.067,-178.643,6.257,148.731
C00626=1181.754,124.541,-53.087,-178.640,6.259,148.730
C00627=1181.749,124.791,-53.106,-178.638,6.261,148.730
C00628=1181.744,125.040,-53.126,-178.635,6.262,148.729
C00629=1181.739,125.289,-53.146,-178.632,6.263,148.729
C00630=1181.734,125.538,-53.166,-178.630,6.265,148.729
C00631=1181.730,125.788,-53.185,-178.628,6.266,148.728
C00632=1181.725,126.037,-53.205,-178.624,6.267,148.728
C00633=1181.720,126.286,-53.225,-178.622,6.269,148.727
C00634=1181.716,126.535,-53.244,-178.619,6.271,148.727
C00635=1181.711,126.784,-53.264,-178.617,6.272,148.726
C00636=1181.706,127.033,-53.284,-178.614,6.273,148.726
C00637=1181.701,127.282,-53.303,-178.611,6.275,148.725
C00638=1181.697,127.532,-53.323,-178.609,6.276,148.725
C00639=1181.692,127.781,-53.343,-178.606,6.278,148.725
C00640=1181.687,128.030,-53.363,-178.603,6.279,148.724
C00641=1181.682,128.279,-53.383,-178.600,6.281,148.724
C00642=1181.678,128.528,-53.403,-178.598,6.282,148.723
C00643=1181.673,128.778,-53.422,-178.596,6.283,148.723
C00644=1181.669,129.027,-53.443,-178.592,6.285,148.722
C00645=1181.663,129.275,-53.462,-178.590,6.287,148.722
C00646=1181.658,129.525,-53.483,-178.588,6.287,148.721
C00647=1181.653,129.774,-53.503,-178.585,6.289,148.721
C00648=1181.649,130.023,-53.523,-178.582,6.291,148.720
C00649=1181.644,130.273,-53.543,-178.580,6.292,148.720
C00650=1181.639,130.522,-53.562,-178.577,6.293,148.720
C00651=1181.634,130.771,-53.582,-178.574,6.295,148.719
C00652=1181.630,131.020,-53.602,-178.571,6.296,148.719
C00653=1181.625,131.269,-53.622,-178.569,6.297,148.718
C00654=1181.620,131.519,-53.642,-178.566,6.299,148.718
C00655=1181.615,131.767,-53.662,-178.563,6.301,148.717
C00656=1181.611,132.016,-53.682,-178.561,6.303,148.717
C00657=1181.605,132.285,-53.704,-178.558,6.304,148.716
C00658=1181.600,132.554,-53.725,-178.555,6.306,148.716
C00659=1181.595,132.822,-53.748,-178.552,6.307,148.715
C00660=1181.590,133.091,-53.769,-178.549,6.309,148.715
C00661=1181.585,133.340,-53.790,-178.547,6.310,148.715
C00662=1181.580,133.589,-53.809,-178.544,6.312,148.714
C00663=1181.576,133.838,-53.830,-178.541,6.313,148.714
C00664=1181.571,134.088,-53.849,-178.538,6.315,148.713
C00665=1181.567,134.337,-53.870,-178.536,6.316,148.713
C00666=1181.561,134.585,-53.890,-178.533,6.317,148.712
C00667=1181.556,134.835,-53.910,-178.531,6.319,148.712
C00668=1181.552,135.084,-53.930,-178.528,6.321,148.711
C00669=1181.547,135.333,-53.951,-178.525,6.322,148.711
C00670=1181.542,135.582,-53.970,-178.523,6.323,148.711
C00671=1181.537,135.832,-53.991,-178.520,6.325,148.710
C00672=1181.533,136.081,-54.012,-178.517,6.327,148.710
C00673=1181.528,136.330,-54.032,-178.514,6.328,148.709
C00674=1181.524,136.579,-54.052,-178.512,6.329,148.709
C00675=1181.518,136.828,-54.073,-178.509,6.331,148.708
C00676=1181.513,137.077,-54.093,-178.507,6.333,148.708
C00677=1181.509,137.326,-54.113,-178.504,6.334,148.708
C00678=1181.504,137.575,-54.133,-178.501,6.336,148.707
C00679=1181.499,137.824,-54.154,-178.499,6.337,148.707
C00680=1181.495,138.073,-54.174,-178.496,6.338,148.706
C00681=1181.490,138.322,-54.194,-178.493,6.340,148.706
C00682=1181.485,138.572,-54.215,-178.491,6.342,148.705
C00683=1181.480,138.821,-54.235,-178.487,6.343,148.705
C00684=1181.476,139.070,-54.255,-178.485,6.344,148.704
C00685=1181.471,139.319,-54.276,-178.483,6.346,148.704
C00686=1181.466,139.568,-54.297,-178.480,6.348,148.704
C00687=1181.462,139.817,-54.317,-178.477,6.350,148.703
C00688=1181.457,140.066,-54.338,-178.475,6.351,148.703
C00689=1181.452,140.315,-54.358,-178.472,6.352,148.702
C00690=1181.448,140.564,-54.379,-178.469,6.354,148.702
C00691=1181.442,140.814,-54.399,-178.467,6.355,148.702
C00692=1181.438,141.063,-54.419,-178.464,6.357,148.701
C00693=1181.433,141.312,-54.440,-178.461,6.359,148.701
C00694=1181.428,141.561,-54.461,-178.458,6.361,148.700
C00695=1181.424,141.810,-54.481,-178.456,6.361,148.700
C00696=1181.419,142.060,-54.502,-178.453,6.363,148.699
C00697=1181.414,142.309,-54.523,-178.450,6.365,148.699
C00698=1181.410,142.558,-54.543,-178.448,6.367,148.699
C00699=1181.405,142.807,-54.564,-178.445,6.368,148.698
C00700=1181.400,143.056,-54.584,-178.442,6.370,148.698
C00701=1181.395,143.305,-54.605,-178.440,6.371,148.697
C00702=1181.390,143.554,-54.626,-178.437,6.372,148.697
C00703=1181.385,143.803,-54.647,-178.434,6.374,148.696
C00704=1181.381,144.052,-54.667,-178.432,6.376,148.696
C00705=1181.376,144.301,-54.688,-178.429,6.378,148.696
C00706=1181.371,144.550,-54.708,-178.426,6.379,148.695
C00707=1181.367,144.799,-54.729,-178.424,6.380,148.695
C00708=1181.362,145.048,-54.750,-178.421,6.382,148.694
C00709=1181.358,145.297,-54.771,-178.418,6.384,148.694
C00710=1181.353,145.547,-54.792,-178.416,6.385,148.694
C00711=1181.348,145.796,-54.813,-178.413,6.387,148.693
C00712=1181.343,146.045,-54.833,-178.410,6.389,148.693
C00713=1181.338,146.294,-54.854,-178.408,6.390,148.692
C00714=1181.334,146.543,-54.875,-178.405,6.391,148.692
C00715=1181.329,146.792,-54.896,-178.402,6.393,148.691
C00716=1181.324,147.041,-54.917,-178.400,6.395,148.691
C00717=1181.319,147.290,-54.938,-178.397,6.396,148.691
C00718=1181.315,147.539,-54.958,-178.394,6.398,148.690
C00719=1181.310,147.788,-54.979,-178.392,6.400,148.690
C00720=1181.306,148.037,-55.000,-178.389,6.402,148.689
C00721=1181.301,148.287,-55.021,-178.387,6.403,148.689
C00722=1181.296,148.536,-55.042,-178.384,6.404,148.689
C00723=1181.291,148.785,-55.063,-178.381,6.406,148.688
C00724=1181.286,149.033,-55.084,-178.378,6.408,148.688
C00725=1181.281,149.283,-55.105,-178.376,6.409,148.687
C00726=1181.277,149.532,-55.126,-178.373,6.411,148.687
C00727=1181.272,149.782,-55.147,-178.370,6.413,148.687
C00728=1181.268,150.030,-55.168,-178.368,6.414,148.686
C00729=1181.263,150.279,-55.189,-178.365,6.416,148.686
C00730=1181.258,150.529,-55.210,-178.363,6.417,148.685
C00731=1181.254,150.777,-55.231,-178.360,6.419,148.685
C00732=1181.248,151.026,-55.252,-178.357,6.421,148.685
C00733=1181.244,151.276,-55.274,-178.354,6.422,148.684
C00734=1181.240,151.524,-55.295,-178.351,6.424,148.684
C00735=1181.235,151.774,-55.316,-178.349,6.426,148.683
C00736=1181.230,152.022,-55.337,-178.346,6.428,148.683
C00737=1181.225,152.272,-55.358,-178.344,6.428,148.683
C00738=1181.221,152.521,-55.379,-178.341,6.430,148.682
C00739=1181.216,152.770,-55.401,-178.339,6.432,148.682
C00740=1181.211,153.019,-55.422,-178.336,6.434,148.681
C00741=1181.207,153.267,-55.443,-178.333,6.436,148.681
C00742=1181.201,153.517,-55.464,-178.330,6.437,148.681
C00743=1181.197,153.766,-55.486,-178.328,6.439,148.680
C00744=1181.192,154.015,-55.507,-178.325,6.440,148.680
C00745=1181.188,154.264,-55.528,-178.322,6.442,148.679
C00746=1181.183,154.513,-55.549,-178.319,6.444,148.679
C00747=1181.178,154.762,-55.571,-178.317,6.445,148.679
C00748=1181.173,155.011,-55.592,-178.314,6.447,148.678
C00749=1181.168,155.260,-55.613,-178.312,6.448,148.678
C00750=1181.164,155.509,-55.634,-178.309,6.450,148.677
C00751=1181.160,155.758,-55.656,-178.306,6.452,148.677
C00752=1181.154,156.008,-55.677,-178.304,6.454,148.677
C00753=1181.150,156.256,-55.699,-178.301,6.456,148.676
C00754=1181.144,156.506,-55.719,-178.298,6.457,148.676
C00755=1181.140,156.755,-55.742,-178.296,6.459,148.676
C00756=1181.136,157.003,-55.763,-178.293,6.461,148.675
C00757=1181.131,157.252,-55.784,-178.290,6.463,148.675
C00758=1181.127,157.502,-55.806,-178.287,6.464,148.674
C00759=1181.121,157.751,-55.827,-178.284,6.466,148.674
C00760=1181.116,158.000,-55.848,-178.282,6.467,148.673
C00761=1181.112,158.269,-55.871,-178.279,6.469,148.673
C00762=1181.107,158.538,-55.895,-178.276,6.471,148.673
C00763=1181.102,158.807,-55.918,-178.274,6.473,148.672
C00764=1181.096,159.076,-55.941,-178.271,6.474,148.672
C00765=1181.091,159.325,-55.963,-178.268,6.476,148.671
C00766=1181.087,159.574,-55.985,-178.265,6.478,148.671
C00767=1181.082,159.823,-56.006,-178.262,6.480,148.671
C00768=1181.077,160.072,-56.028,-178.260,6.481,148.670
C00769=1181.074,160.321,-56.049,-178.257,6.483,148.670
C00770=1181.069,160.569,-56.071,-178.254,6.485,148.669
C00771=1181.064,160.819,-56.092,-178.252,6.487,148.669
C00772=1181.059,161.068,-56.114,-178.249,6.488,148.669
C00773=1181.054,161.317,-56.135,-178.246,6.490,148.668
C00774=1181.050,161.565,-56.157,-178.244,6.492,148.668
C00775=1181.045,161.815,-56.179,-178.241,6.494,148.668
C00776=1181.040,162.063,-56.201,-178.238,6.495,148.667
C00777=1181.036,162.313,-56.222,-178.236,6.497,148.667
C00778=1181.031,162.562,-56.244,-178.233,6.499,148.666
C00779=1181.026,162.811,-56.266,-178.230,6.501,148.666
C00780=1181.022,163.060,-56.288,-178.228,6.502,148.666
C00781=1181.017,163.309,-56.309,-178.225,6.504,148.665
C00782=1181.013,163.558,-56.331,-178.223,6.505,148.665
C00783=1181.008,163.807,-56.353,-178.220,6.507,148.665
C00784=1181.003,164.055,-56.375,-178.217,6.509,148.664
C00785=1180.998,164.305,-56.397,-178.215,6.511,148.664
C00786=1180.993,164.554,-56.418,-178.212,6.512,148.664
C00787=1180.989,164.803,-56.440,-178.209,6.514,148.663
C00788=1180.984,165.052,-56.462,-178.207,6.516,148.663
C00789=1180.979,165.301,-56.484,-178.204,6.518,148.662
C00790=1180.975,165.550,-56.506,-178.201,6.519,148.662
C00791=1180.970,165.799,-56.528,-178.199,6.521,148.662
C00792=1180.965,166.048,-56.550,-178.196,6.523,148.661
C00793=1180.961,166.297,-56.572,-178.193,6.525,148.661
C00794=1180.956,166.546,-56.593,-178.191,6.527,148.661
C00795=1180.951,166.795,-56.615,-178.188,6.528,148.660
C00796=1180.946,167.044,-56.638,-178.185,6.530,148.660
C00797=1180.942,167.292,-56.660,-178.183,6.532,148.659
C00798=1180.938,167.542,-56.682,-178.180,6.534,148.659
C00799=1180.933,167.790,-56.704,-178.177,6.535,148.659
C00800=1180.928,168.040,-56.726,-178.175,6.537,148.658
C00801=1180.924,168.288,-56.747,-178.172,6.539,148.658
C00802=1180.919,168.538,-56.770,-178.169,6.541,148.658
C00803=1180.914,168.787,-56.792,-178.166,6.542,148.657
C00804=1180.909,169.036,-56.814,-178.164,6.544,148.657
C00805=1180.905,169.285,-56.835,-178.161,6.546,148.657
C00806=1180.900,169.534,-56.859,-178.158,6.548,148.656
C00807=1180.895,169.782,-56.881,-178.156,6.550,148.656
C00808=1180.891,170.032,-56.903,-178.153,6.551,148.655
C00809=1180.886,170.281,-56.925,-178.150,6.553,148.655
C00810=1180.881,170.530,-56.947,-178.148,6.555,148.655
C00811=1180.877,170.779,-56.970,-178.145,6.557,148.654
C00812=1180.872,171.027,-56.991,-178.142,6.558,148.654
C00813=1180.868,171.277,-57.013,-178.140,6.560,148.654
C00814=1180.862,171.526,-57.036,-178.137,6.562,148.653
C00815=1180.858,171.775,-57.058,-178.134,6.564,148.653
C00816=1180.853,172.023,-57.080,-178.132,6.566,148.652
C00817=1180.849,172.272,-57.102,-178.128,6.568,148.652
C00818=1180.844,172.522,-57.125,-178.126,6.570,148.652
C00819=1180.839,172.770,-57.147,-178.123,6.572,148.651
C00820=1180.835,173.019,-57.169,-178.120,6.573,148.651
C00821=1180.830,173.268,-57.192,-178.118,6.576,148.651
C00822=1180.826,173.517,-57.214,-178.115,6.577,148.651
C00823=1180.821,173.766,-57.236,-178.113,6.579,148.650
C00824=1180.816,174.015,-57.259,-178.110,6.581,148.650
C00825=1180.812,174.264,-57.281,-178.107,6.583,148.649
C00826=1180.806,174.513,-57.304,-178.105,6.584,148.649
C00827=1180.802,174.762,-57.326,-178.102,6.586,148.649
C00828=1180.798,175.011,-57.348,-178.099,6.588,148.648
C00829=1180.792,175.260,-57.371,-178.097,6.590,148.648
C00830=1180.788,175.509,-57.394,-178.094,6.592,148.648
C00831=1180.784,175.758,-57.416,-178.091,6.593,148.647
C00832=1180.779,176.006,-57.439,-178.089,6.595,148.647
C00833=1180.775,176.256,-57.461,-178.086,6.597,148.647
C00834=1180.770,176.505,-57.484,-178.083,6.599,148.646
C00835=1180.765,176.753,-57.506,-178.081,6.600,148.646
C00836=1180.760,177.002,-57.529,-178.078,6.603,148.646
C00837=1180.756,177.252,-57.551,-178.075,6.605,148.645
C00838=1180.751,177.500,-57.574,-178.073,6.607,148.645
C00839=1180.746,177.749,-57.596,-178.070,6.609,148.645
C00840=1180.742,177.998,-57.619,-178.067,6.611,148.644
C00841=1180.737,178.247,-57.641,-178.065,6.612,148.644
C00842=1180.733,178.496,-57.664,-178.062,6.614,148.644
C00843=1180.728,178.745,-57.687,-178.059,6.616,148.643
C00844=1180.723,178.993,-57.709,-178.057,6.618,148.643
C00845=1180.719,179.242,-57.732,-178.054,6.619,148.642
C00846=1180.714,179.492,-57.754,-178.051,6.621,148.642
C00847=1180.710,179.741,-57.778,-178.048,6.623,148.642
C00848=1180.705,179.989,-57.799,-178.046,6.625,148.642
C00849=1180.700,180.238,-57.823,-178.044,6.627,148.641
C00850=1180.695,180.488,-57.846,-178.040,6.629,148.641
C00851=1180.691,180.737,-57.868,-178.038,6.631,148.641
C00852=1180.686,180.985,-57.891,-178.035,6.633,148.640
C00853=1180.682,181.234,-57.914,-178.032,6.635,148.640
C00854=1180.677,181.484,-57.937,-178.030,6.637,148.639
C00855=1180.673,181.732,-57.959,-178.027,6.638,148.639
C00856=1180.668,181.981,-57.982,-178.024,6.640,148.639
C00857=1180.663,182.230,-58.006,-178.022,6.642,148.639
C00858=1180.659,182.479,-58.028,-178.019,6.644,148.638
C00859=1180.654,182.728,-58.051,-178.017,6.646,148.638
C00860=1180.649,182.976,-58.073,-178.014,6.648,148.638
C00861=1180.645,183.225,-58.097,-178.011,6.650,148.637
C00862=1180.640,183.475,-58.119,-178.008,6.652,148.637
C00863=1180.636,183.723,-58.142,-178.006,6.654,148.636
C00864=1180.631,183.972,-58.166,-178.003,6.656,148.636
C00865=1180.626,184.242,-58.191,-178.000,6.657,148.636
C00866=1180.621,184.512,-58.215,-177.997,6.660,148.635
C00867=1180.616,184.781,-58.240,-177.994,6.662,148.635
C00868=1180.610,185.051,-58.265,-177.992,6.664,148.635
C00869=1180.606,185.299,-58.288,-177.988,6.666,148.634
C00870=1180.601,185.548,-58.311,-177.986,6.668,148.634
C00871=1180.596,185.797,-58.334,-177.983,6.670,148.634
C00872=1180.593,186.046,-58.357,-177.981,6.672,148.634
C00873=1180.588,186.295,-58.380,-177.978,6.674,148.633
C00874=1180.583,186.544,-58.404,-177.975,6.675,148.633
C00875=1180.578,186.793,-58.427,-177.973,6.677,148.632
C00876=1180.574,187.041,-58.450,-177.970,6.680,148.632
C00877=1180.569,187.290,-58.473,-177.967,6.682,148.632
C00878=1180.564,187.539,-58.496,-177.965,6.684,148.632
C00879=1180.560,187.788,-58.520,-177.962,6.685,148.631
C00880=1180.556,188.037,-58.542,-177.959,6.687,148.631
C00881=1180.551,188.286,-58.566,-177.957,6.689,148.631
C00882=1180.546,188.535,-58.589,-177.954,6.691,148.630
C00883=1180.542,188.784,-58.612,-177.951,6.694,148.630
C00884=1180.536,189.032,-58.635,-177.949,6.696,148.630
C00885=1180.532,189.281,-58.658,-177.946,6.697,148.629
C00886=1180.528,189.530,-58.682,-177.943,6.699,148.629
C00887=1180.523,189.779,-58.705,-177.941,6.701,148.629
C00888=1180.518,190.028,-58.728,-177.938,6.703,148.628
C00889=1180.514,190.277,-58.752,-177.936,6.705,148.628
C00890=1180.509,190.526,-58.775,-177.932,6.707,148.628
C00891=1180.505,190.775,-58.798,-177.930,6.709,148.628
C00892=1180.501,191.023,-58.822,-177.927,6.711,148.627
C00893=1180.496,191.272,-58.845,-177.924,6.713,148.627
C00894=1180.491,191.521,-58.869,-177.922,6.715,148.627
C00895=1180.486,191.771,-58.892,-177.920,6.717,148.626
C00896=1180.482,192.020,-58.915,-177.916,6.719,148.626
C00897=1180.477,192.269,-58.939,-177.914,6.721,148.626
C00898=1180.472,192.516,-58.962,-177.911,6.723,148.625
C00899=1180.467,192.765,-58.986,-177.908,6.725,148.625
C00900=1180.463,193.014,-59.009,-177.906,6.727,148.625
C00901=1180.458,193.263,-59.032,-177.903,6.729,148.625
C00902=1180.453,193.512,-59.056,-177.900,6.731,148.624
C00903=1180.449,193.761,-59.080,-177.898,6.733,148.624
C00904=1180.445,194.010,-59.103,-177.895,6.735,148.623
C00905=1180.440,194.259,-59.126,-177.893,6.737,148.623
C00906=1180.436,194.507,-59.150,-177.890,6.739,148.623
C00907=1180.431,194.756,-59.173,-177.887,6.741,148.623
C00908=1180.426,195.005,-59.197,-177.884,6.743,148.622
C00909=1180.422,195.253,-59.221,-177.881,6.745,148.622
C00910=1180.417,195.503,-59.244,-177.879,6.747,148.622
C00911=1180.413,195.752,-59.268,-177.877,6.749,148.622
C00912=1180.408,196.000,-59.292,-177.873,6.751,148.621
C00913=1180.403,196.250,-59.316,-177.871,6.753,148.621
C00914=1180.399,196.499,-59.339,-177.868,6.755,148.621
C00915=1180.394,196.747,-59.363,-177.866,6.757,148.620
C00916=1180.390,196.996,-59.387,-177.863,6.759,148.620
C00917=1180.385,197.245,-59.411,-177.860,6.762,148.620
C00918=1180.381,197.494,-59.434,-177.857,6.763,148.619
C00919=1180.376,197.743,-59.458,-177.855,6.765,148.619
C00920=1180.371,197.991,-59.482,-177.852,6.767,148.619
C00921=1180.367,198.240,-59.505,-177.850,6.769,148.619
C00922=1180.362,198.489,-59.529,-177.846,6.772,148.618
C00923=1180.358,198.738,-59.552,-177.844,6.774,148.618
C00924=1180.353,198.986,-59.576,-177.842,6.776,148.618
C00925=1180.348,199.236,-59.600,-177.839,6.777,148.617
C00926=1180.343,199.484,-59.624,-177.836,6.779,148.617
C00927=1180.339,199.734,-59.648,-177.834,6.782,148.617
C00928=1180.335,199.982,-59.672,-177.831,6.784,148.617
C00929=1180.331,200.231,-59.696,-177.828,6.786,148.616
C00930=1180.326,200.480,-59.720,-177.826,6.787,148.616
C00931=1180.321,200.728,-59.744,-177.823,6.790,148.616
C00932=1180.316,200.977,-59.768,-177.820,6.792,148.615
C00933=1180.312,201.226,-59.792,-177.817,6.794,148.615
C00934=1180.307,201.474,-59.816,-177.815,6.796,148.615
C00935=1180.303,201.724,-59.840,-177.812,6.799,148.615
C00936=1180.299,201.972,-59.864,-177.809,6.801,148.614
C00937=1180.294,202.221,-59.888,-177.807,6.802,148.614
C00938=1180.289,202.470,-59.912,-177.804,6.804,148.614
C00939=1180.284,202.718,-59.936,-177.801,6.807,148.614
C00940=1180.280,202.967,-59.960,-177.799,6.809,148.613
C00941=1180.275,203.217,-59.984,-177.796,6.811,148.613
C00942=1180.271,203.465,-60.008,-177.793,6.812,148.612
C00943=1180.266,203.714,-60.032,-177.791,6.815,148.612
C00944=1180.262,203.963,-60.056,-177.788,6.817,148.612
C00945=1180.257,204.212,-60.080,-177.785,6.819,148.612
C00946=1180.253,204.461,-60.105,-177.783,6.821,148.612
C00947=1180.248,204.709,-60.129,-177.780,6.824,148.611
C00948=1180.244,204.957,-60.153,-177.777,6.826,148.611
C00949=1180.239,205.207,-60.177,-177.774,6.827,148.611
C00950=1180.234,205.455,-60.201,-177.772,6.829,148.610
C00951=1180.230,205.704,-60.225,-177.769,6.832,148.610
C00952=1180.225,205.953,-60.250,-177.766,6.834,148.610
C00953=1180.221,206.201,-60.274,-177.764,6.836,148.610
C00954=1180.216,206.451,-60.298,-177.762,6.838,148.609
C00955=1180.212,206.700,-60.323,-177.758,6.840,148.609
C00956=1180.207,206.948,-60.347,-177.756,6.843,148.609
C00957=1180.202,207.197,-60.371,-177.753,6.844,148.609
C00958=1180.198,207.445,-60.395,-177.750,6.847,148.608
C00959=1180.194,207.695,-60.420,-177.748,6.849,148.608
C00960=1180.189,207.943,-60.444,-177.745,6.851,148.608
C00961=1180.184,208.192,-60.469,-177.743,6.853,148.607
C00962=1180.179,208.440,-60.493,-177.739,6.855,148.607
C00963=1180.176,208.690,-60.518,-177.737,6.857,148.607
C00964=1180.171,208.938,-60.542,-177.735,6.859,148.607
C00965=1180.166,209.187,-60.566,-177.731,6.862,148.606
C00966=1180.162,209.436,-60.591,-177.729,6.864,148.606
C00967=1180.157,209.685,-60.616,-177.727,6.866,148.606
C00968=1180.153,209.933,-60.640,-177.724,6.868,148.606
C00969=1180.147,210.204,-60.666,-177.721,6.870,148.605
C00970=1180.143,210.475,-60.693,-177.718,6.873,148.605
C00971=1180.138,210.745,-60.719,-177.715,6.875,148.605
C00972=1180.132,211.015,-60.746,-177.712,6.878,148.604
C00973=1180.129,211.264,-60.771,-177.709,6.879,148.604
C00974=1180.123,211.513,-60.795,-177.707,6.882,148.604
C00975=1180.119,211.761,-60.819,-177.704,6.884,148.604
C00976=1180.115,212.011,-60.844,-177.701,6.886,148.603
C00977=1180.110,212.259,-60.870,-177.699,6.888,148.603
C00978=1180.105,212.507,-60.894,-177.696,6.891,148.603
C00979=1180.101,212.757,-60.919,-177.693,6.892,148.603
C00980=1180.096,213.005,-60.943,-177.691,6.895,148.603
C00981=1180.091,213.254,-60.968,-177.688,6.897,148.602
C00982=1180.087,213.503,-60.992,-177.685,6.899,148.602
C00983=1180.083,213.751,-61.017,-177.683,6.901,148.602
C00984=1180.079,214.000,-61.042,-177.680,6.904,148.601
C00985=1180.074,214.249,-61.067,-177.677,6.906,148.601
C00986=1180.069,214.497,-61.091,-177.675,6.908,148.601
C00987=1180.065,214.747,-61.116,-177.672,6.910,148.601
C00988=1180.060,214.995,-61.141,-177.669,6.913,148.601
C00989=1180.055,215.244,-61.166,-177.667,6.914,148.600
C00990=1180.051,215.493,-61.190,-177.664,6.916,148.600
C00991=1180.046,215.741,-61.215,-177.661,6.919,148.600
C00992=1180.042,215.990,-61.240,-177.659,6.921,148.599
C00993=1180.037,216.238,-61.265,-177.656,6.923,148.599
C00994=1180.033,216.487,-61.290,-177.653,6.926,148.599
C00995=1180.029,216.736,-61.314,-177.651,6.927,148.599
C00996=1180.024,216.985,-61.339,-177.648,6.930,148.599
C00997=1180.019,217.233,-61.365,-177.645,6.932,148.598
C00998=1180.015,217.483,-61.390,-177.643,6.934,148.598
C00999=1180.010,217.731,-61.414,-177.640,6.937,148.598
C01000=1180.006,217.979,-61.439,-177.637,6.939,148.598
C01001=1180.001,218.229,-61.464,-177.635,6.941,148.597
C01002=1179.997,218.476,-61.489,-177.632,6.944,148.597
C01003=1179.992,218.726,-61.514,-177.629,6.945,148.597
C01004=1179.988,218.974,-61.540,-177.627,6.947,148.597
C01005=1179.983,219.223,-61.565,-177.624,6.950,148.596
C01006=1179.979,219.472,-61.589,-177.621,6.952,148.596
C01007=1179.974,219.721,-61.614,-177.619,6.954,148.596
C01008=1179.969,219.969,-61.639,-177.616,6.957,148.596
C01009=1179.965,220.218,-61.665,-177.613,6.959,148.595
C01010=1179.961,220.466,-61.689,-177.611,6.961,148.595
C01011=1179.956,220.715,-61.715,-177.608,6.963,148.595
C01012=1179.952,220.963,-61.740,-177.605,6.965,148.595
C01013=1179.947,221.213,-61.765,-177.602,6.968,148.594
C01014=1179.943,221.462,-61.791,-177.600,6.970,148.594
C01015=1179.938,221.710,-61.816,-177.597,6.972,148.594
C01016=1179.934,221.959,-61.841,-177.595,6.975,148.594
C01017=1179.929,222.208,-61.865,-177.592,6.977,148.594
C01018=1179.925,222.456,-61.891,-177.589,6.978,148.593
C01019=1179.920,222.704,-61.916,-177.587,6.981,148.593
C01020=1179.916,222.954,-61.942,-177.584,6.983,148.593
C01021=1179.911,223.202,-61.967,-177.581,6.986,148.593
C01022=1179.906,223.451,-61.993,-177.578,6.988,148.592
C01023=1179.902,223.700,-62.018,-177.576,6.990,148.592
C01024=1179.898,223.948,-62.042,-177.573,6.993,148.592
C01025=1179.894,224.197,-62.068,-177.570,6.995,148.592
C01026=1179.888,224.446,-62.093,-177.568,6.998,148.592
C01027=1179.884,224.694,-62.119,-177.565,6.999,148.591
C01028=1179.880,224.943,-62.144,-177.563,7.002,148.591
C01029=1179.875,225.191,-62.170,-177.560,7.004,148.591
C01030=1179.871,225.441,-62.195,-177.557,7.006,148.591
C01031=1179.866,225.689,-62.220,-177.554,7.009,148.590
C01032=1179.862,225.938,-62.246,-177.552,7.011,148.590
C01033=1179.857,226.186,-62.272,-177.549,7.013,148.590
C01034=1179.853,226.435,-62.297,-177.547,7.016,148.590
C01035=1179.848,226.684,-62.322,-177.544,7.018,148.590
C01036=1179.844,226.933,-62.348,-177.541,7.021,148.590
C01037=1179.839,227.181,-62.373,-177.539,7.022,148.589
C01038=1179.835,227.430,-62.399,-177.536,7.024,148.589
C01039=1179.830,227.678,-62.424,-177.533,7.027,148.589
C01040=1179.826,227.927,-62.450,-177.531,7.029,148.588
C01041=1179.822,228.175,-62.476,-177.528,7.032,148.588
C01042=1179.817,228.423,-62.501,-177.525,7.034,148.588
C01043=1179.812,228.673,-62.526,-177.522,7.037,148.588
C01044=1179.808,228.922,-62.552,-177.520,7.039,148.588
C01045=1179.804,229.171,-62.578,-177.518,7.041,148.588
C01046=1179.799,229.419,-62.603,-177.514,7.043,148.587
C01047=1179.794,229.668,-62.630,-177.512,7.045,148.587
C01048=1179.790,229.917,-62.655,-177.509,7.048,148.587
C01049=1179.785,230.165,-62.681,-177.507,7.050,148.587
C01050=1179.781,230.413,-62.706,-177.504,7.053,148.586
C01051=1179.776,230.662,-62.732,-177.501,7.055,148.586
C01052=1179.772,230.910,-62.758,-177.499,7.057,148.586
C01053=1179.767,231.159,-62.783,-177.496,7.060,148.586
C01054=1179.763,231.408,-62.809,-177.493,7.062,148.586
C01055=1179.758,231.657,-62.835,-177.491,7.065,148.586
C01056=1179.754,231.905,-62.862,-177.488,7.066,148.585
C01057=1179.749,232.153,-62.887,-177.485,7.069,148.585
C01058=1179.745,232.402,-62.913,-177.483,7.071,148.585
C01059=1179.741,232.651,-62.939,-177.480,7.074,148.585
C01060=1179.736,232.899,-62.964,-177.478,7.076,148.585
C01061=1179.731,233.148,-62.991,-177.475,7.078,148.584
C01062=1179.727,233.397,-63.016,-177.472,7.081,148.584
C01063=1179.723,233.646,-63.042,-177.470,7.083,148.584
C01064=1179.718,233.893,-63.068,-177.467,7.086,148.584
C01065=1179.713,234.142,-63.094,-177.464,7.088,148.583
C01066=1179.709,234.391,-63.120,-177.461,7.091,148.583
C01067=1179.705,234.640,-63.146,-177.459,7.092,148.583
C01068=1179.701,234.889,-63.172,-177.456,7.095,148.583
C01069=1179.695,235.137,-63.198,-177.454,7.097,148.583
C01070=1179.691,235.385,-63.224,-177.451,7.100,148.583
C01071=1179.687,235.634,-63.250,-177.448,7.102,148.583
C01072=1179.683,235.883,-63.276,-177.445,7.105,148.582
C01073=1179.678,236.155,-63.305,-177.443,7.107,148.582
C01074=1179.673,236.427,-63.333,-177.440,7.110,148.582
C01075=1179.668,236.697,-63.361,-177.437,7.112,148.582
C01076=1179.662,236.969,-63.390,-177.434,7.115,148.581
C01077=1179.658,237.217,-63.417,-177.432,7.117,148.581
C01078=1179.654,237.466,-63.442,-177.428,7.120,148.581
C01079=1179.649,237.715,-63.469,-177.426,7.122,148.581
C01080=1179.645,237.964,-63.495,-177.423,7.125,148.581
C01081=1179.641,238.212,-63.520,-177.421,7.127,148.581
C01082=1179.636,238.460,-63.548,-177.418,7.130,148.580
C01083=1179.632,238.709,-63.573,-177.415,7.132,148.580
C01084=1179.627,238.958,-63.600,-177.413,7.135,148.580
C01085=1179.623,239.206,-63.626,-177.410,7.137,148.580
C01086=1179.619,239.455,-63.652,-177.407,7.140,148.580
C01087=1179.614,239.704,-63.679,-177.405,7.141,148.579
C01088=1179.610,239.952,-63.705,-177.402,7.144,148.579
C01089=1179.605,240.201,-63.732,-177.400,7.146,148.579
C01090=1179.600,240.449,-63.757,-177.397,7.149,148.579
C01091=1179.596,240.697,-63.784,-177.394,7.151,148.579
C01092=1179.591,240.946,-63.810,-177.391,7.154,148.579
C01093=1179.587,241.194,-63.836,-177.389,7.156,148.578
C01094=1179.582,241.444,-63.863,-177.386,7.159,148.578
C01095=1179.579,241.692,-63.889,-177.384,7.161,148.578
C01096=1179.574,241.941,-63.916,-177.381,7.164,148.578
C01097=1179.570,242.189,-63.942,-177.379,7.166,148.578
C01098=1179.565,242.438,-63.969,-177.375,7.169,148.578
C01099=1179.561,242.686,-63.995,-177.373,7.171,148.578
C01100=1179.556,242.935,-64.022,-177.371,7.174,148.577
C01101=1179.552,243.184,-64.048,-177.368,7.175,148.577
C01102=1179.547,243.432,-64.075,-177.365,7.178,148.577
C01103=1179.543,243.680,-64.101,-177.363,7.180,148.577
C01104=1179.538,243.929,-64.128,-177.360,7.183,148.577
C01105=1179.534,244.178,-64.155,-177.357,7.186,148.577
C01106=1179.530,244.426,-64.181,-177.354,7.188,148.576
C01107=1179.525,244.675,-64.207,-177.352,7.191,148.576
C01108=1179.521,244.923,-64.234,-177.349,7.193,148.576
C01109=1179.516,245.172,-64.261,-177.346,7.196,148.576
C01110=1179.512,245.420,-64.287,-177.344,7.198,148.576
C01111=1179.507,245.669,-64.314,-177.341,7.201,148.576
C01112=1179.503,245.918,-64.341,-177.339,7.203,148.575
C01113=1179.499,246.166,-64.367,-177.336,7.206,148.575
C01114=1179.494,246.414,-64.394,-177.334,7.208,148.575
C01115=1179.489,246.663,-64.421,-177.331,7.210,148.575
C01116=1179.485,246.912,-64.447,-177.328,7.213,148.575
C01117=1179.481,247.160,-64.474,-177.326,7.216,148.575
C01118=1179.476,247.409,-64.501,-177.322,7.218,148.575
C01119=1179.472,247.657,-64.528,-177.320,7.220,148.574
C01120=1179.467,247.905,-64.555,-177.318,7.223,148.574
C01121=1179.463,248.154,-64.582,-177.315,7.226,148.574
C01122=1179.459,248.402,-64.608,-177.312,7.228,148.574
C01123=1179.454,248.651,-64.635,-177.310,7.230,148.574
C01124=1179.449,248.900,-64.662,-177.307,7.233,148.574
C01125=1179.444,249.148,-64.689,-177.304,7.236,148.574
C01126=1179.441,249.397,-64.716,-177.302,7.238,148.573
C01127=1179.437,249.646,-64.743,-177.299,7.241,148.573
C01128=1179.432,249.894,-64.770,-177.297,7.243,148.573
C01129=1179.428,250.142,-64.796,-177.294,7.246,148.573
C01130=1179.423,250.391,-64.823,-177.292,7.248,148.573
C01131=1179.419,250.639,-64.850,-177.289,7.251,148.573
C01132=1179.414,250.888,-64.877,-177.286,7.254,148.573
C01133=1179.409,251.136,-64.904,-177.283,7.256,148.572
C01134=1179.405,251.384,-64.931,-177.281,7.259,148.572
C01135=1179.401,251.634,-64.958,-177.278,7.261,148.572
C01136=1179.397,251.882,-64.985,-177.275,7.264,148.572
C01137=1179.392,252.131,-65.012,-177.273,7.266,148.572
C01138=1179.388,252.378,-65.040,-177.270,7.269,148.572
C01139=1179.384,252.627,-65.067,-177.268,7.272,148.572
C01140=1179.379,252.875,-65.094,-177.265,7.273,148.572
C01141=1179.375,253.124,-65.121,-177.262,7.276,148.571
C01142=1179.370,253.373,-65.148,-177.260,7.279,148.571
C01143=1179.366,253.621,-65.175,-177.257,7.282,148.571
C01144=1179.361,253.870,-65.202,-177.254,7.284,148.571
C01145=1179.357,254.118,-65.230,-177.252,7.286,148.571
C01146=1179.352,254.366,-65.257,-177.249,7.289,148.571
C01147=1179.349,254.615,-65.284,-177.246,7.292,148.571
C01148=1179.344,254.864,-65.311,-177.244,7.294,148.570
C01149=1179.339,255.112,-65.338,-177.241,7.297,148.570
C01150=1179.335,255.360,-65.366,-177.239,7.299,148.570
C01151=1179.330,255.608,-65.393,-177.236,7.302,148.570
C01152=1179.326,255.858,-65.420,-177.233,7.305,148.570
C01153=1179.322,256.106,-65.448,-177.231,7.307,148.570
C01154=1179.317,256.354,-65.475,-177.228,7.310,148.570
C01155=1179.313,256.603,-65.502,-177.226,7.312,148.570
C01156=1179.309,256.852,-65.530,-177.223,7.315,148.570
C01157=1179.304,257.100,-65.558,-177.220,7.318,148.569
C01158=1179.300,257.348,-65.585,-177.218,7.320,148.569
C01159=1179.295,257.597,-65.612,-177.215,7.323,148.569
C01160=1179.291,257.845,-65.640,-177.212,7.326,148.569
C01161=1179.287,258.094,-65.667,-177.210,7.328,148.569
C01162=1179.282,258.342,-65.694,-177.207,7.331,148.569
C01163=1179.278,258.590,-65.722,-177.205,7.333,148.569
C01164=1179.274,258.839,-65.749,-177.202,7.336,148.569
C01165=1179.269,259.087,-65.777,-177.199,7.339,148.569
C01166=1179.265,259.336,-65.804,-177.197,7.341,148.569
C01167=1179.261,259.584,-65.832,-177.194,7.344,148.568
C01168=1179.256,259.833,-65.859,-177.191,7.347,148.568
C01169=1179.252,260.081,-65.887,-177.189,7.349,148.568
C01170=1179.247,260.329,-65.914,-177.186,7.352,148.568
C01171=1179.243,260.578,-65.943,-177.184,7.355,148.568
C01172=1179.238,260.826,-65.970,-177.181,7.357,148.568
C01173=1179.234,261.074,-65.998,-177.178,7.359,148.568
C01174=1179.230,261.324,-66.025,-177.175,7.362,148.568
C01175=1179.225,261.571,-66.053,-177.173,7.365,148.568
C01176=1179.221,261.820,-66.080,-177.171,7.368,148.568
C01177=1179.216,262.093,-66.111,-177.168,7.370,148.567
C01178=1179.211,262.367,-66.141,-177.165,7.373,148.567
C01179=1179.206,262.639,-66.172,-177.162,7.376,148.567
C01180=1179.201,262.912,-66.202,-177.159,7.379,148.567
C01181=1179.197,263.160,-66.230,-177.156,7.382,148.567
C01182=1179.193,263.409,-66.258,-177.154,7.384,148.567
C01183=1179.189,263.657,-66.285,-177.151,7.387,148.567
C01184=1179.184,263.905,-66.313,-177.148,7.390,148.567
C01185=1179.180,264.154,-66.342,-177.146,7.392,148.567
C01186=1179.175,264.403,-66.369,-177.143,7.395,148.566
C01187=1179.171,264.651,-66.397,-177.141,7.398,148.566
C01188=1179.167,264.899,-66.425,-177.138,7.400,148.566
C01189=1179.162,265.147,-66.453,-177.136,7.403,148.566
C01190=1179.158,265.397,-66.480,-177.132,7.406,148.566
C01191=1179.153,265.644,-66.508,-177.130,7.408,148.566
C01192=1179.150,265.893,-66.536,-177.128,7.411,148.566
C01193=1179.145,266.141,-66.565,-177.125,7.414,148.566
C01194=1179.140,266.390,-66.592,-177.123,7.416,148.566
C01195=1179.136,266.638,-66.620,-177.120,7.419,148.566
C01196=1179.131,266.886,-66.648,-177.117,7.422,148.566
C01197=1179.127,267.135,-66.677,-177.114,7.425,148.566
C01198=1179.123,267.383,-66.704,-177.112,7.427,148.566
C01199=1179.119,267.632,-66.733,-177.109,7.430,148.565
C01200=1179.114,267.880,-66.760,-177.106,7.433,148.565
C01201=1179.110,268.129,-66.788,-177.104,7.435,148.565
C01202=1179.105,268.377,-66.817,-177.101,7.438,148.565
C01203=1179.101,268.625,-66.844,-177.099,7.441,148.565
C01204=1179.096,268.874,-66.873,-177.097,7.443,148.565
C01205=1179.092,269.122,-66.901,-177.094,7.446,148.565
C01206=1179.088,269.370,-66.929,-177.091,7.449,148.565
C01207=1179.083,269.618,-66.957,-177.088,7.452,148.565
C01208=1179.079,269.867,-66.986,-177.086,7.454,148.565
C01209=1179.074,270.115,-67.014,-177.083,7.457,148.565
C01210=1179.070,270.364,-67.042,-177.080,7.460,148.564
C01211=1179.066,270.612,-67.070,-177.078,7.462,148.564
C01212=1179.062,270.861,-67.099,-177.075,7.465,148.564
C01213=1179.058,271.109,-67.127,-177.073,7.468,148.564
C01214=1179.053,271.357,-67.155,-177.070,7.471,148.564
C01215=1179.049,271.606,-67.183,-177.068,7.473,148.564
C01216=1179.044,271.854,-67.212,-177.065,7.476,148.564
C01217=1179.040,272.103,-67.240,-177.062,7.479,148.564
C01218=1179.035,272.351,-67.268,-177.060,7.481,148.564
C01219=1179.032,272.599,-67.297,-177.057,7.484,148.564
C01220=1179.027,272.847,-67.325,-177.055,7.487,148.564
C01221=1179.023,273.096,-67.353,-177.052,7.490,148.564
C01222=1179.018,273.344,-67.382,-177.050,7.492,148.564
C01223=1179.014,273.592,-67.410,-177.047,7.495,148.564
C01224=1179.009,273.841,-67.439,-177.044,7.498,148.564
C01225=1179.005,274.088,-67.467,-177.042,7.501,148.564
C01226=1179.001,274.337,-67.496,-177.039,7.503,148.564
C01227=1178.997,274.585,-67.524,-177.037,7.506,148.563
C01228=1178.992,274.834,-67.552,-177.034,7.509,148.563
C01229=1178.988,275.083,-67.581,-177.031,7.512,148.563
C01230=1178.984,275.330,-67.610,-177.029,7.514,148.563
C01231=1178.979,275.579,-67.638,-177.026,7.517,148.563
C01232=1178.975,275.828,-67.667,-177.023,7.520,148.563
C01233=1178.971,276.075,-67.696,-177.020,7.523,148.563
C01234=1178.966,276.324,-67.724,-177.018,7.525,148.563
C01235=1178.962,276.572,-67.752,-177.015,7.528,148.563
C01236=1178.958,276.820,-67.782,-177.013,7.531,148.563
C01237=1178.953,277.069,-67.810,-177.010,7.534,148.563
C01238=1178.949,277.317,-67.838,-177.008,7.536,148.563
C01239=1178.944,277.565,-67.868,-177.005,7.539,148.563
C01240=1178.941,277.814,-67.896,-177.002,7.542,148.563
C01241=1178.936,278.062,-67.924,-177.000,7.545,148.563
C01242=1178.931,278.310,-67.954,-176.997,7.547,148.562
C01243=1178.927,278.559,-67.982,-176.995,7.550,148.562
C01244=1178.924,278.807,-68.011,-176.992,7.553,148.562
C01245=1178.918,279.055,-68.040,-176.989,7.556,148.562
C01246=1178.914,279.304,-68.069,-176.987,7.558,148.562
C01247=1178.911,279.552,-68.097,-176.984,7.561,148.562
C01248=1178.906,279.800,-68.126,-176.982,7.564,148.562
C01249=1178.901,280.049,-68.155,-176.979,7.568,148.562
C01250=1178.897,280.297,-68.184,-176.977,7.571,148.562
C01251=1178.893,280.546,-68.213,-176.974,7.573,148.562
C01252=1178.889,280.793,-68.242,-176.972,7.576,148.562
C01253=1178.884,281.042,-68.270,-176.969,7.579,148.562
C01254=1178.880,281.290,-68.300,-176.966,7.582,148.562
C01255=1178.875,281.538,-68.328,-176.964,7.584,148.562
C01256=1178.871,281.786,-68.357,-176.961,7.587,148.562
C01257=1178.867,282.035,-68.387,-176.959,7.590,148.562
C01258=1178.863,282.284,-68.415,-176.956,7.593,148.562
C01259=1178.858,282.531,-68.444,-176.953,7.596,148.562
C01260=1178.853,282.780,-68.473,-176.951,7.598,148.562
C01261=1178.849,283.028,-68.503,-176.948,7.601,148.562
C01262=1178.846,283.276,-68.531,-176.946,7.604,148.562
C01263=1178.842,283.524,-68.561,-176.943,7.607,148.562
C01264=1178.837,283.773,-68.589,-176.940,7.610,148.562
C01265=1178.832,284.021,-68.619,-176.938,7.612,148.562
C01266=1178.828,284.269,-68.648,-176.935,7.615,148.562
C01267=1178.824,284.518,-68.677,-176.932,7.618,148.562
C01268=1178.819,284.766,-68.706,-176.930,7.621,148.562
C01269=1178.815,285.014,-68.735,-176.927,7.624,148.561
C01270=1178.811,285.262,-68.765,-176.925,7.627,148.562
C01271=1178.806,285.511,-68.794,-176.923,7.630,148.562
C01272=1178.803,285.759,-68.822,-176.920,7.633,148.562
C01273=1178.798,286.007,-68.852,-176.917,7.636,148.562
C01274=1178.794,286.255,-68.881,-176.914,7.638,148.561
C01275=1178.789,286.503,-68.910,-176.912,7.641,148.561
C01276=1178.785,286.751,-68.940,-176.909,7.644,148.561
C01277=1178.781,287.000,-68.969,-176.907,7.647,148.561
C01278=1178.777,287.249,-68.998,-176.904,7.650,148.561
C01279=1178.772,287.497,-69.028,-176.901,7.653,148.561
C01280=1178.768,287.745,-69.057,-176.899,7.655,148.561
C01281=1178.763,288.019,-69.090,-176.896,7.659,148.561
C01282=1178.758,288.295,-69.123,-176.893,7.662,148.561
C01283=1178.753,288.569,-69.154,-176.890,7.665,148.561
C01284=1178.749,288.844,-69.188,-176.888,7.668,148.561
C01285=1178.744,289.092,-69.217,-176.885,7.671,148.561
C01286=1178.740,289.340,-69.246,-176.883,7.674,148.561
C01287=1178.736,289.588,-69.276,-176.880,7.677,148.561
C01288=1178.732,289.837,-69.305,-176.877,7.680,148.561
C01289=1178.727,290.084,-69.334,-176.874,7.683,148.561
C01290=1178.723,290.333,-69.364,-176.872,7.685,148.561
C01291=1178.719,290.581,-69.393,-176.870,7.688,148.561
C01292=1178.715,290.829,-69.423,-176.867,7.691,148.561
C01293=1178.710,291.077,-69.452,-176.865,7.694,148.561
C01294=1178.705,291.326,-69.482,-176.862,7.697,148.561
C01295=1178.701,291.574,-69.512,-176.859,7.700,148.561
C01296=1178.697,291.822,-69.541,-176.857,7.702,148.561
C01297=1178.693,292.070,-69.571,-176.854,7.705,148.561
C01298=1178.689,292.318,-69.601,-176.851,7.708,148.561
C01299=1178.685,292.567,-69.630,-176.849,7.711,148.561
C01300=1178.680,292.815,-69.660,-176.846,7.714,148.561
C01301=1178.676,293.064,-69.690,-176.844,7.718,148.561
C01302=1178.672,293.312,-69.719,-176.842,7.720,148.561
C01303=1178.668,293.559,-69.749,-176.839,7.723,148.561
C01304=1178.663,293.808,-69.779,-176.836,7.726,148.561
C01305=1178.659,294.056,-69.809,-176.833,7.729,148.561
C01306=1178.654,294.305,-69.838,-176.831,7.732,148.561
C01307=1178.651,294.552,-69.869,-176.828,7.735,148.561
C01308=1178.646,294.800,-69.898,-176.826,7.738,148.561
C01309=1178.642,295.049,-69.927,-176.823,7.740,148.561
C01310=1178.637,295.297,-69.957,-176.821,7.743,148.561
C01311=1178.633,295.545,-69.988,-176.818,7.746,148.561
C01312=1178.629,295.793,-70.017,-176.815,7.749,148.561
C01313=1178.624,296.042,-70.047,-176.813,7.752,148.561
C01314=1178.620,296.289,-70.077,-176.810,7.755,148.561
C01315=1178.616,296.538,-70.107,-176.808,7.758,148.561
C01316=1178.612,296.785,-70.137,-176.805,7.761,148.561
C01317=1178.607,297.034,-70.167,-176.803,7.764,148.561
C01318=1178.603,297.282,-70.196,-176.800,7.767,148.561
C01319=1178.599,297.530,-70.227,-176.798,7.770,148.561
C01320=1178.595,297.779,-70.257,-176.795,7.773,148.561
C01321=1178.591,298.027,-70.287,-176.792,7.776,148.561
C01322=1178.587,298.275,-70.317,-176.790,7.779,148.561
C01323=1178.582,298.523,-70.347,-176.787,7.782,148.561
C01324=1178.578,298.771,-70.377,-176.785,7.784,148.561
C01325=1178.574,299.019,-70.408,-176.782,7.787,148.561
C01326=1178.569,299.267,-70.437,-176.780,7.790,148.561
C01327=1178.566,299.515,-70.467,-176.777,7.793,148.561
C01328=1178.561,299.764,-70.497,-176.775,7.797,148.561
C01329=1178.557,300.011,-70.527,-176.772,7.800,148.561
C01330=1178.552,300.261,-70.558,-176.769,7.803,148.561
C01331=1178.549,300.508,-70.588,-176.766,7.805,148.561
C01332=1178.544,300.757,-70.618,-176.765,7.808,148.561
C01333=1178.540,301.005,-70.648,-176.762,7.811,148.561
C01334=1178.535,301.252,-70.679,-176.759,7.814,148.561
C01335=1178.531,301.501,-70.708,-176.757,7.817,148.561
C01336=1178.527,301.748,-70.739,-176.754,7.820,148.562
C01337=1178.523,301.997,-70.770,-176.752,7.823,148.562
C01338=1178.519,302.245,-70.799,-176.749,7.826,148.561
C01339=1178.514,302.493,-70.830,-176.746,7.829,148.561
C01340=1178.510,302.741,-70.861,-176.744,7.833,148.562
C01341=1178.505,302.989,-70.890,-176.742,7.835,148.562
C01342=1178.501,303.237,-70.921,-176.739,7.838,148.562
C01343=1178.498,303.486,-70.952,-176.736,7.841,148.562
C01344=1178.493,303.734,-70.982,-176.734,7.844,148.562
C01345=1178.489,303.982,-71.012,-176.731,7.847,148.562
C01346=1178.484,304.230,-71.043,-176.729,7.850,148.562
C01347=1178.480,304.478,-71.073,-176.726,7.853,148.562
C01348=1178.476,304.726,-71.104,-176.724,7.856,148.562
C01349=1178.471,304.975,-71.134,-176.721,7.859,148.562
C01350=1178.467,305.223,-71.164,-176.718,7.862,148.562
C01351=1178.463,305.470,-71.195,-176.715,7.865,148.562
C01352=1178.459,305.718,-71.225,-176.714,7.868,148.562
C01353=1178.455,305.967,-71.256,-176.711,7.871,148.562
C01354=1178.450,306.215,-71.287,-176.708,7.874,148.562
C01355=1178.446,306.462,-71.317,-176.706,7.877,148.562
C01356=1178.442,306.711,-71.347,-176.703,7.880,148.562
C01357=1178.438,306.960,-71.378,-176.700,7.883,148.562
C01358=1178.434,307.207,-71.408,-176.698,7.886,148.562
C01359=1178.429,307.455,-71.439,-176.696,7.889,148.562
C01360=1178.424,307.703,-71.470,-176.693,7.892,148.562
C01361=1178.421,307.952,-71.500,-176.690,7.895,148.562
C01362=1178.417,308.199,-71.531,-176.688,7.899,148.562
C01363=1178.412,308.447,-71.562,-176.685,7.902,148.562
C01364=1178.408,308.696,-71.593,-176.683,7.904,148.562
C01365=1178.404,308.944,-71.623,-176.681,7.907,148.563
C01366=1178.399,309.192,-71.654,-176.678,7.910,148.562
C01367=1178.395,309.440,-71.685,-176.675,7.913,148.562
C01368=1178.391,309.688,-71.716,-176.673,7.916,148.563
C01369=1178.387,309.936,-71.746,-176.670,7.919,148.563
C01370=1178.383,310.185,-71.777,-176.667,7.922,148.563
C01371=1178.379,310.432,-71.809,-176.665,7.926,148.563
C01372=1178.374,310.680,-71.839,-176.662,7.929,148.563
C01373=1178.371,310.928,-71.870,-176.660,7.932,148.563
C01374=1178.366,311.176,-71.901,-176.657,7.935,148.563
C01375=1178.362,311.424,-71.932,-176.655,7.938,148.563
C01376=1178.358,311.673,-71.963,-176.652,7.941,148.563
C01377=1178.353,311.921,-71.993,-176.650,7.944,148.563
C01378=1178.349,312.168,-72.025,-176.647,7.947,148.563
C01379=1178.345,312.417,-72.055,-176.645,7.950,148.563
C01380=1178.341,312.664,-72.086,-176.643,7.953,148.563
C01381=1178.336,312.912,-72.117,-176.640,7.956,148.563
C01382=1178.332,313.160,-72.149,-176.638,7.959,148.563
C01383=1178.328,313.408,-72.180,-176.635,7.962,148.563
C01384=1178.324,313.657,-72.211,-176.632,7.965,148.563
C01385=1178.319,313.933,-72.245,-176.629,7.969,148.564
C01386=1178.314,314.210,-72.279,-176.627,7.972,148.564
C01387=1178.310,314.487,-72.314,-176.624,7.975,148.564
C01388=1178.305,314.764,-72.349,-176.621,7.979,148.564
C01389=1178.301,315.012,-72.381,-176.618,7.982,148.564
C01390=1178.296,315.260,-72.412,-176.616,7.985,148.564
C01391=1178.292,315.508,-72.443,-176.613,7.988,148.564
C01392=1178.288,315.756,-72.473,-176.611,7.991,148.564
C01393=1178.284,316.003,-72.505,-176.608,7.995,148.564
C01394=1178.280,316.252,-72.536,-176.606,7.998,148.564
C01395=1178.276,316.499,-72.567,-176.603,8.001,148.564
C01396=1178.272,316.748,-72.599,-176.601,8.003,148.564
C01397=1178.267,316.995,-72.630,-176.598,8.006,148.564
C01398=1178.263,317.244,-72.661,-176.596,8.010,148.565
C01399=1178.259,317.492,-72.692,-176.594,8.013,148.565
C01400=1178.255,317.740,-72.724,-176.591,8.016,148.565
C01401=1178.251,317.988,-72.754,-176.589,8.019,148.565
C01402=1178.247,318.236,-72.786,-176.586,8.022,148.565
C01403=1178.243,318.483,-72.818,-176.584,8.025,148.565
C01404=1178.238,318.732,-72.850,-176.581,8.028,148.565
C01405=1178.233,318.980,-72.881,-176.579,8.031,148.565
C01406=1178.229,319.228,-72.912,-176.576,8.034,148.565
C01407=1178.225,319.476,-72.944,-176.574,8.038,148.565
C01408=1178.221,319.724,-72.975,-176.571,8.041,148.565
C01409=1178.217,319.972,-73.006,-176.569,8.044,148.565
C01410=1178.213,320.220,-73.038,-176.566,8.047,148.565
C01411=1178.209,320.468,-73.069,-176.564,8.050,148.566
C01412=1178.205,320.716,-73.101,-176.561,8.053,148.566
C01413=1178.201,320.963,-73.132,-176.559,8.057,148.566
C01414=1178.196,321.212,-73.164,-176.556,8.060,148.566
C01415=1178.192,321.460,-73.196,-176.554,8.063,148.566
C01416=1178.188,321.707,-73.227,-176.551,8.066,148.566
C01417=1178.184,321.956,-73.258,-176.549,8.069,148.566
C01418=1178.179,322.203,-73.290,-176.546,8.072,148.566
C01419=1178.176,322.451,-73.322,-176.544,8.076,148.566
C01420=1178.171,322.699,-73.353,-176.541,8.079,148.566
C01421=1178.167,322.948,-73.385,-176.539,8.082,148.567
C01422=1178.163,323.196,-73.417,-176.536,8.085,148.567
C01423=1178.159,323.443,-73.448,-176.534,8.088,148.567
C01424=1178.155,323.691,-73.480,-176.531,8.091,148.567
C01425=1178.150,323.939,-73.512,-176.529,8.094,148.567
C01426=1178.146,324.187,-73.544,-176.526,8.097,148.567
C01427=1178.142,324.435,-73.575,-176.524,8.101,148.567
C01428=1178.138,324.683,-73.607,-176.521,8.104,148.567
C01429=1178.134,324.931,-73.638,-176.519,8.107,148.567
C01430=1178.130,325.179,-73.671,-176.516,8.110,148.568
C01431=1178.125,325.426,-73.702,-176.514,8.113,148.568
C01432=1178.122,325.674,-73.734,-176.511,8.117,148.568
C01433=1178.117,325.923,-73.767,-176.509,8.120,148.568
C01434=1178.113,326.170,-73.798,-176.506,8.123,148.568
C01435=1178.109,326.418,-73.830,-176.504,8.126,148.568
C01436=1178.105,326.667,-73.862,-176.501,8.129,148.568
C01437=1178.100,326.914,-73.894,-176.499,8.132,148.568
C01438=1178.097,327.162,-73.926,-176.496,8.136,148.568
C01439=1178.092,327.410,-73.958,-176.494,8.139,148.569
C01440=1178.088,327.658,-73.990,-176.491,8.142,148.569
C01441=1178.084,327.906,-74.021,-176.489,8.145,148.569
C01442=1178.080,328.154,-74.054,-176.486,8.148,148.569
C01443=1178.076,328.401,-74.085,-176.484,8.151,148.569
C01444=1178.072,328.649,-74.117,-176.482,8.155,148.569
C01445=1178.067,328.898,-74.150,-176.479,8.158,148.569
C01446=1178.064,329.146,-74.182,-176.477,8.161,148.569
C01447=1178.059,329.393,-74.214,-176.474,8.164,148.569
C01448=1178.055,329.641,-74.245,-176.472,8.167,148.570
C01449=1178.051,329.890,-74.278,-176.470,8.171,148.570
C01450=1178.047,330.137,-74.310,-176.467,8.174,148.570
C01451=1178.043,330.385,-74.342,-176.465,8.177,148.570
C01452=1178.038,330.633,-74.374,-176.462,8.180,148.570
C01453=1178.035,330.881,-74.406,-176.460,8.183,148.570
C01454=1178.030,331.129,-74.438,-176.457,8.187,148.570
C01455=1178.026,331.376,-74.471,-176.455,8.190,148.571
C01456=1178.022,331.624,-74.503,-176.452,8.193,148.571
C01457=1178.018,331.872,-74.535,-176.450,8.196,148.571
C01458=1178.014,332.121,-74.568,-176.448,8.200,148.571
C01459=1178.010,332.367,-74.600,-176.445,8.203,148.571
C01460=1178.005,332.616,-74.632,-176.443,8.206,148.571
C01461=1178.001,332.864,-74.664,-176.441,8.209,148.572
C01462=1177.997,333.112,-74.697,-176.438,8.212,148.572
C01463=1177.992,333.359,-74.729,-176.436,8.215,148.572
C01464=1177.989,333.607,-74.761,-176.433,8.219,148.572
C01465=1177.984,333.855,-74.794,-176.431,8.222,148.572
C01466=1177.981,334.103,-74.826,-176.428,8.225,148.572
C01467=1177.976,334.351,-74.859,-176.426,8.228,148.572
C01468=1177.973,334.599,-74.891,-176.424,8.232,148.573
C01469=1177.968,334.846,-74.923,-176.421,8.236,148.573
C01470=1177.964,335.094,-74.956,-176.418,8.239,148.573
C01471=1177.960,335.342,-74.988,-176.416,8.242,148.573
C01472=1177.956,335.591,-75.021,-176.414,8.245,148.573
C01473=1177.951,335.838,-75.054,-176.411,8.248,148.573
C01474=1177.948,336.086,-75.086,-176.409,8.252,148.573
C01475=1177.944,336.334,-75.119,-176.407,8.255,148.574
C01476=1177.939,336.582,-75.151,-176.404,8.258,148.574
C01477=1177.935,336.829,-75.183,-176.402,8.261,148.574
C01478=1177.931,337.078,-75.216,-176.399,8.265,148.574
C01479=1177.927,337.325,-75.249,-176.397,8.268,148.574
C01480=1177.923,337.573,-75.282,-176.395,8.271,148.575
C01481=1177.919,337.821,-75.314,-176.392,8.275,148.575
C01482=1177.915,338.069,-75.347,-176.390,8.278,148.575
C01483=1177.911,338.317,-75.379,-176.387,8.281,148.575
C01484=1177.907,338.565,-75.412,-176.385,8.284,148.575
C01485=1177.902,338.812,-75.444,-176.383,8.288,148.575
C01486=1177.898,339.060,-75.477,-176.381,8.291,148.576
C01487=1177.894,339.307,-75.510,-176.378,8.294,148.576
C01488=1177.890,339.556,-75.542,-176.376,8.297,148.576
C01489=1177.885,339.835,-75.580,-176.373,8.301,148.576
C01490=1177.881,340.114,-75.617,-176.370,8.305,148.576
C01491=1177.875,340.393,-75.654,-176.368,8.309,148.577
C01492=1177.872,340.672,-75.691,-176.365,8.313,148.577
C01493=1177.867,340.920,-75.724,-176.362,8.316,148.577
C01494=1177.863,341.168,-75.756,-176.360,8.319,148.577
C01495=1177.859,341.416,-75.789,-176.358,8.322,148.577
C01496=1177.855,341.663,-75.823,-176.355,8.326,148.577
C01497=1177.851,341.911,-75.855,-176.353,8.329,148.578
C01498=1177.847,342.159,-75.888,-176.351,8.332,148.578
C01499=1177.843,342.407,-75.921,-176.349,8.336,148.578
C01500=1177.839,342.655,-75.954,-176.346,8.339,148.578
C01501=1177.834,342.902,-75.987,-176.344,8.342,148.579
C01502=1177.830,343.150,-76.020,-176.341,8.346,148.579
C01503=1177.826,343.398,-76.053,-176.339,8.349,148.579
C01504=1177.822,343.646,-76.086,-176.336,8.353,148.579
C01505=1177.818,343.894,-76.118,-176.334,8.356,148.579
C01506=1177.814,344.141,-76.151,-176.332,8.359,148.579
C01507=1177.810,344.389,-76.185,-176.329,8.363,148.580
C01508=1177.806,344.637,-76.218,-176.327,8.366,148.580
C01509=1177.802,344.885,-76.251,-176.325,8.369,148.580
C01510=1177.798,345.132,-76.284,-176.323,8.373,148.580
C01511=1177.794,345.380,-76.317,-176.320,8.376,148.580
C01512=1177.789,345.628,-76.350,-176.318,8.379,148.581
C01513=1177.785,345.875,-76.384,-176.316,8.383,148.581
C01514=1177.781,346.123,-76.417,-176.313,8.387,148.581
C01515=1177.777,346.371,-76.450,-176.311,8.390,148.581
C01516=1177.773,346.619,-76.483,-176.308,8.393,148.582
C01517=1177.769,346.866,-76.516,-176.306,8.397,148.582
C01518=1177.765,347.114,-76.549,-176.304,8.400,148.582
C01519=1177.760,347.362,-76.582,-176.302,8.403,148.582
C01520=1177.756,347.610,-76.616,-176.299,8.407,148.582
C01521=1177.752,347.857,-76.649,-176.297,8.410,148.583
C01522=1177.748,348.104,-76.683,-176.295,8.413,148.583
C01523=1177.745,348.353,-76.716,-176.293,8.416,148.583
C01524=1177.741,348.601,-76.749,-176.290,8.421,148.584
C01525=1177.736,348.849,-76.783,-176.288,8.424,148.584
C01526=1177.732,349.096,-76.816,-176.286,8.428,148.584
C01527=1177.727,349.344,-76.849,-176.283,8.431,148.584
C01528=1177.724,349.591,-76.883,-176.281,8.434,148.584
C01529=1177.720,349.839,-76.916,-176.279,8.437,148.585
C01530=1177.715,350.087,-76.950,-176.277,8.441,148.585
C01531=1177.712,350.335,-76.983,-176.274,8.444,148.585
C01532=1177.708,350.582,-77.017,-176.272,8.447,148.585
C01533=1177.704,350.830,-77.050,-176.270,8.452,148.586
C01534=1177.699,351.078,-77.084,-176.267,8.455,148.586
C01535=1177.695,351.326,-77.117,-176.265,8.458,148.586
C01536=1177.691,351.573,-77.151,-176.263,8.462,148.586
C01537=1177.687,351.821,-77.184,-176.261,8.465,148.587
C01538=1177.683,352.069,-77.218,-176.258,8.468,148.587
C01539=1177.679,352.316,-77.252,-176.256,8.472,148.587
C01540=1177.675,352.564,-77.285,-176.254,8.475,148.588
C01541=1177.671,352.812,-77.318,-176.252,8.479,148.588
C01542=1177.667,353.059,-77.352,-176.249,8.483,148.588
C01543=1177.663,353.307,-77.386,-176.247,8.486,148.588
C01544=1177.659,353.555,-77.420,-176.245,8.490,148.589
C01545=1177.654,353.803,-77.453,-176.243,8.493,148.589
C01546=1177.650,354.050,-77.487,-176.240,8.496,148.589
C01547=1177.647,354.298,-77.521,-176.238,8.500,148.589
C01548=1177.642,354.546,-77.555,-176.236,8.503,148.590
C01549=1177.638,354.793,-77.588,-176.233,8.507,148.590
C01550=1177.634,355.041,-77.622,-176.231,8.511,148.590
C01551=1177.631,355.289,-77.656,-176.229,8.514,148.591
C01552=1177.626,355.537,-77.690,-176.227,8.518,148.591
C01553=1177.622,355.784,-77.723,-176.225,8.521,148.591
C01554=1177.618,356.032,-77.757,-176.223,8.524,148.591
C01555=1177.614,356.280,-77.791,-176.221,8.528,148.592
C01556=1177.610,356.527,-77.825,-176.218,8.532,148.592
C01557=1177.606,356.775,-77.858,-176.216,8.535,148.592
C01558=1177.602,357.022,-77.893,-176.214,8.539,148.593
C01559=1177.598,357.270,-77.926,-176.212,8.542,148.593
C01560=1177.594,357.518,-77.960,-176.210,8.546,148.593
C01561=1177.590,357.765,-77.995,-176.207,8.549,148.594
C01562=1177.586,358.013,-78.028,-176.205,8.552,148.594
C01563=1177.582,358.260,-78.062,-176.203,8.557,148.594
C01564=1177.578,358.508,-78.097,-176.201,8.560,148.595
C01565=1177.574,358.756,-78.130,-176.199,8.564,148.595
C01566=1177.570,359.004,-78.165,-176.196,8.567,148.595
C01567=1177.566,359.251,-78.198,-176.194,8.570,148.595
C01568=1177.561,359.499,-78.232,-176.192,8.574,148.596
C01569=1177.558,359.747,-78.266,-176.190,8.577,148.596
C01570=1177.554,359.994,-78.300,-176.188,8.582,148.597
C01571=1177.550,360.242,-78.335,-176.185,8.585,148.597
C01572=1177.546,360.489,-78.369,-176.184,8.589,148.597
C01573=1177.541,360.737,-78.403,-176.182,8.592,148.598
C01574=1177.538,360.985,-78.437,-176.179,8.596,148.598
C01575=1177.533,361.232,-78.472,-176.178,8.599,148.598
C01576=1177.530,361.479,-78.505,-176.175,8.603,148.598
C01577=1177.526,361.728,-78.540,-176.174,8.606,148.599
C01578=1177.522,361.975,-78.574,-176.172,8.610,148.599
C01579=1177.517,362.223,-78.608,-176.169,8.613,148.600
C01580=1177.514,362.471,-78.642,-176.167,8.618,148.600
C01581=1177.509,362.718,-78.677,-176.165,8.621,148.600
C01582=1177.506,362.966,-78.711,-176.163,8.624,148.601
C01583=1177.501,363.213,-78.745,-176.161,8.628,148.601
C01584=1177.497,363.460,-78.779,-176.159,8.632,148.602
C01585=1177.493,363.708,-78.814,-176.157,8.635,148.602
C01586=1177.490,363.956,-78.848,-176.155,8.639,148.602
C01587=1177.486,364.204,-78.883,-176.153,8.642,148.603
C01588=1177.481,364.451,-78.917,-176.152,8.646,148.603
C01589=1177.478,364.699,-78.951,-176.150,8.649,148.603
C01590=1177.473,364.946,-78.986,-176.148,8.653,148.604
C01591=1177.470,365.194,-79.020,-176.146,8.657,148.604
C01592=1177.466,365.442,-79.055,-176.144,8.660,148.605
C01593=1177.461,365.723,-79.094,-176.141,8.664,148.605
C01594=1177.456,366.004,-79.133,-176.140,8.668,148.606
C01595=1177.452,366.287,-79.172,-176.138,8.673,148.606
C01596=1177.448,366.569,-79.211,-176.136,8.676,148.607
C01597=1177.443,366.816,-79.245,-176.134,8.680,148.607
C01598=1177.440,367.064,-79.281,-176.132,8.684,148.607
C01599=1177.435,367.311,-79.315,-176.130,8.687,148.608
C01600=1177.432,367.559,-79.350,-176.128,8.691,148.608
C01601=1177.427,367.806,-79.384,-176.127,8.694,148.609
C01602=1177.423,368.054,-79.419,-176.125,8.698,148.609
C01603=1177.419,368.302,-79.453,-176.123,8.702,148.610
C01604=1177.416,368.549,-79.488,-176.121,8.705,148.610
C01605=1177.411,368.796,-79.523,-176.119,8.709,148.610
C01606=1177.408,369.044,-79.557,-176.118,8.713,148.611
C01607=1177.403,369.292,-79.591,-176.116,8.716,148.612
C01608=1177.399,369.540,-79.626,-176.114,8.720,148.612
C01609=1177.395,369.787,-79.661,-176.113,8.723,148.612
C01610=1177.392,370.034,-79.696,-176.112,8.727,148.613
C01611=1177.387,370.282,-79.730,-176.110,8.730,148.613
C01612=1177.383,370.530,-79.765,-176.108,8.734,148.614
C01613=1177.379,370.777,-79.800,-176.106,8.738,148.614
C01614=1177.375,371.025,-79.835,-176.105,8.742,148.615
C01615=1177.371,371.272,-79.869,-176.103,8.744,148.615
C01616=1177.368,371.520,-79.904,-176.102,8.748,148.616
C01617=1177.364,371.768,-79.939,-176.100,8.752,148.616
C01618=1177.359,372.015,-79.974,-176.098,8.755,148.617
C01619=1177.355,372.263,-80.009,-176.097,8.759,148.617
C01620=1177.352,372.510,-80.043,-176.096,8.762,148.618
C01621=1177.348,372.757,-80.079,-176.094,8.766,148.618
C01622=1177.343,373.005,-80.113,-176.093,8.770,148.619
C01623=1177.339,373.253,-80.148,-176.091,8.774,148.620
C01624=1177.336,373.500,-80.184,-176.090,8.776,148.620
C01625=1177.331,373.748,-80.218,-176.088,8.780,148.621
C01626=1177.328,373.995,-80.253,-176.087,8.784,148.621
C01627=1177.324,374.242,-80.287,-176.086,8.787,148.622
C01628=1177.320,374.490,-80.323,-176.084,8.791,148.622
C01629=1177.316,374.738,-80.358,-176.083,8.795,148.623
C01630=1177.311,374.985,-80.392,-176.082,8.798,148.623
C01631=1177.308,375.233,-80.428,-176.080,8.802,148.624
C01632=1177.303,375.480,-80.462,-176.079,8.804,148.624
C01633=1177.300,375.728,-80.498,-176.078,8.808,148.625
C01634=1177.296,375.976,-80.533,-176.076,8.812,148.625
C01635=1177.292,376.222,-80.567,-176.075,8.815,148.626
C01636=1177.288,376.470,-80.603,-176.074,8.819,148.627
C01637=1177.284,376.717,-80.637,-176.073,8.822,148.627
C01638=1177.280,376.965,-80.673,-176.071,8.826,148.628
C01639=1177.276,377.213,-80.708,-176.071,8.829,148.628
C01640=1177.272,377.460,-80.743,-176.069,8.833,148.629
C01641=1177.268,377.708,-80.778,-176.068,8.836,148.629
C01642=1177.264,377.955,-80.813,-176.067,8.840,148.630
C01643=1177.260,378.202,-80.848,-176.066,8.843,148.631
C01644=1177.256,378.450,-80.883,-176.064,8.847,148.631
C01645=1177.252,378.698,-80.919,-176.063,8.850,148.632
C01646=1177.248,378.944,-80.954,-176.063,8.853,148.632
C01647=1177.244,379.193,-80.989,-176.061,8.857,148.633
C01648=1177.241,379.440,-81.024,-176.060,8.860,148.633
C01649=1177.236,379.687,-81.059,-176.060,8.863,148.634
C01650=1177.232,379.935,-81.094,-176.058,8.867,148.635
C01651=1177.229,380.183,-81.130,-176.057,8.870,148.635
C01652=1177.224,380.429,-81.165,-176.057,8.873,148.636
C01653=1177.220,380.677,-81.200,-176.056,8.877,148.637
C01654=1177.217,380.925,-81.235,-176.055,8.880,148.637
C01655=1177.212,381.172,-81.271,-176.054,8.883,148.638
C01656=1177.208,381.420,-81.305,-176.053,8.887,148.638
C01657=1177.205,381.667,-81.341,-176.052,8.890,148.639
C01658=1177.201,381.915,-81.377,-176.051,8.894,148.640
C01659=1177.196,382.162,-81.412,-176.050,8.897,148.640
C01660=1177.192,382.410,-81.447,-176.050,8.900,148.641
C01661=1177.189,382.658,-81.483,-176.049,8.903,148.642
C01662=1177.184,382.904,-81.518,-176.048,8.906,148.642
C01663=1177.181,383.152,-81.553,-176.047,8.910,148.643
C01664=1177.177,383.399,-81.589,-176.046,8.914,148.644
C01665=1177.173,383.648,-81.624,-176.045,8.917,148.644
C01666=1177.169,383.894,-81.659,-176.045,8.920,148.645
C01667=1177.165,384.142,-81.695,-176.044,8.923,148.645
C01668=1177.161,384.389,-81.730,-176.043,8.926,148.646
C01669=1177.157,384.636,-81.765,-176.042,8.929,148.647
C01670=1177.153,384.884,-81.801,-176.042,8.933,148.647
C01671=1177.149,385.132,-81.836,-176.041,8.936,148.648
C01672=1177.145,385.380,-81.872,-176.041,8.939,148.649
C01673=1177.141,385.626,-81.907,-176.041,8.941,148.649
C01674=1177.137,385.874,-81.943,-176.040,8.945,148.650
C01675=1177.133,386.121,-81.978,-176.039,8.948,148.651
C01676=1177.130,386.369,-82.014,-176.039,8.951,148.651
C01677=1177.125,386.616,-82.049,-176.038,8.954,148.652
C01678=1177.121,386.863,-82.085,-176.037,8.957,148.653
C01679=1177.117,387.111,-82.120,-176.037,8.960,148.653
C01680=1177.114,387.358,-82.156,-176.037,8.963,148.654
C01681=1177.110,387.607,-82.191,-176.036,8.967,148.655
C01682=1177.106,387.853,-82.226,-176.035,8.970,148.655
C01683=1177.101,388.101,-82.262,-176.036,8.972,148.656
C01684=1177.098,388.349,-82.298,-176.035,8.976,148.657
C01685=1177.094,388.596,-82.333,-176.034,8.979,148.657
C01686=1177.090,388.843,-82.368,-176.035,8.981,148.658
C01687=1177.086,389.090,-82.404,-176.034,8.984,148.659
C01688=1177.082,389.338,-82.440,-176.034,8.987,148.659
C01689=1177.078,389.586,-82.476,-176.033,8.990,148.660
C01690=1177.074,389.833,-82.511,-176.033,8.993,148.661
C01691=1177.070,390.080,-82.546,-176.033,8.996,148.661
C01692=1177.066,390.328,-82.582,-176.032,8.999,148.662
C01693=1177.063,390.575,-82.618,-176.032,9.002,148.663
C01694=1177.058,390.823,-82.654,-176.032,9.005,148.663
C01695=1177.055,391.070,-82.689,-176.031,9.007,148.664
C01696=1177.050,391.317,-82.724,-176.032,9.010,148.665
C01697=1177.046,391.602,-82.766,-176.031,9.013,148.666
C01698=1177.042,391.886,-82.807,-176.031,9.017,148.666
C01699=1177.037,392.171,-82.848,-176.030,9.020,148.667
C01700=1177.032,392.455,-82.888,-176.031,9.023,148.668
C01701=1177.029,392.702,-82.924,-176.030,9.026,148.669
C01702=1177.024,392.950,-82.960,-176.030,9.029,148.669
C01703=1177.021,393.198,-82.996,-176.031,9.031,148.670
C01704=1177.017,393.445,-83.031,-176.030,9.034,148.671
C01705=1177.013,393.691,-83.067,-176.030,9.037,148.671
C01706=1177.009,393.939,-83.103,-176.030,9.039,148.672
C01707=1177.005,394.187,-83.139,-176.030,9.042,148.673
C01708=1177.001,394.434,-83.174,-176.029,9.045,148.673
C01709=1176.998,394.682,-83.210,-176.030,9.048,148.674
C01710=1176.993,394.929,-83.246,-176.029,9.050,148.675
C01711=1176.989,395.176,-83.281,-176.029,9.052,148.675
C01712=1176.985,395.424,-83.317,-176.030,9.055,148.676
C01713=1176.981,395.671,-83.353,-176.029,9.058,148.677
C01714=1176.978,395.918,-83.389,-176.029,9.061,148.677
C01715=1176.974,396.166,-83.425,-176.029,9.063,148.678
C01716=1176.969,396.414,-83.461,-176.029,9.066,148.679
C01717=1176.965,396.660,-83.496,-176.029,9.068,148.679
C01718=1176.962,396.908,-83.532,-176.029,9.071,148.680
C01719=1176.958,397.155,-83.567,-176.029,9.073,148.681
C01720=1176.953,397.403,-83.603,-176.029,9.076,148.681
C01721=1176.950,397.650,-83.639,-176.029,9.078,148.682
C01722=1176.946,397.898,-83.675,-176.029,9.081,148.683
C01723=1176.942,398.145,-83.711,-176.030,9.083,148.683
C01724=1176.938,398.392,-83.746,-176.029,9.085,148.684
C01725=1176.934,398.640,-83.782,-176.029,9.088,148.685
C01726=1176.930,398.888,-83.818,-176.030,9.091,148.685
C01727=1176.926,399.134,-83.854,-176.030,9.093,148.686
C01728=1176.923,399.382,-83.890,-176.029,9.095,148.687
C01729=1176.918,399.630,-83.926,-176.030,9.098,148.687
C01730=1176.915,399.877,-83.962,-176.030,9.100,148.688
C01731=1176.910,400.124,-83.997,-176.030,9.103,148.688
C01732=1176.906,400.371,-84.034,-176.030,9.105,148.689
C01733=1176.903,400.619,-84.069,-176.030,9.107,148.690
C01734=1176.899,400.866,-84.105,-176.030,9.109,148.690
C01735=1176.895,401.114,-84.141,-176.030,9.112,148.691
C01736=1176.891,401.362,-84.176,-176.030,9.114,148.692
C01737=1176.888,401.608,-84.213,-176.030,9.117,148.692
C01738=1176.883,401.856,-84.249,-176.030,9.119,148.693
C01739=1176.879,402.103,-84.284,-176.031,9.121,148.694
C01740=1176.874,402.351,-84.320,-176.031,9.123,148.694
C01741=1176.871,402.598,-84.356,-176.031,9.126,148.695
C01742=1176.867,402.845,-84.392,-176.031,9.128,148.695
C01743=1176.863,403.093,-84.428,-176.031,9.130,148.696
C01744=1176.859,403.341,-84.464,-176.032,9.132,148.697
C01745=1176.856,403.587,-84.500,-176.031,9.135,148.697
C01746=1176.852,403.835,-84.536,-176.032,9.137,148.698
C01747=1176.848,404.083,-84.572,-176.032,9.139,148.699
C01748=1176.843,404.330,-84.607,-176.032,9.141,148.699
C01749=1176.840,404.577,-84.644,-176.032,9.144,148.700
C01750=1176.836,404.824,-84.679,-176.032,9.145,148.700
C01751=1176.832,405.072,-84.715,-176.033,9.148,148.701
C01752=1176.828,405.319,-84.752,-176.032,9.150,148.702
C01753=1176.825,405.566,-84.787,-176.033,9.152,148.702
C01754=1176.820,405.814,-84.823,-176.033,9.154,148.703
C01755=1176.816,406.062,-84.859,-176.033,9.157,148.704
C01756=1176.812,406.309,-84.896,-176.034,9.158,148.704
C01757=1176.808,406.556,-84.931,-176.033,9.161,148.705
C01758=1176.804,406.803,-84.966,-176.034,9.163,148.705
C01759=1176.800,407.050,-85.003,-176.034,9.165,148.706
C01760=1176.797,407.298,-85.039,-176.034,9.167,148.707
C01761=1176.792,407.546,-85.075,-176.034,9.169,148.707
C01762=1176.789,407.793,-85.111,-176.034,9.171,148.708
C01763=1176.785,408.040,-85.147,-176.034,9.174,148.708
C01764=1176.781,408.288,-85.183,-176.035,9.175,148.709
C01765=1176.778,408.535,-85.219,-176.035,9.178,148.709
C01766=1176.773,408.783,-85.255,-176.035,9.179,148.710
C01767=1176.769,409.030,-85.291,-176.035,9.182,148.711
C01768=1176.766,409.277,-85.327,-176.035,9.183,148.711
C01769=1176.761,409.524,-85.363,-176.036,9.186,148.712
C01770=1176.757,409.772,-85.398,-176.036,9.187,148.712
C01771=1176.753,410.019,-85.435,-176.036,9.190,148.713
C01772=1176.750,410.266,-85.471,-176.036,9.191,148.713
C01773=1176.745,410.514,-85.507,-176.036,9.193,148.714
C01774=1176.742,410.761,-85.543,-176.037,9.195,148.715
C01775=1176.738,411.008,-85.579,-176.036,9.197,148.715
C01776=1176.734,411.256,-85.615,-176.037,9.199,148.716
C01777=1176.730,411.503,-85.651,-176.037,9.201,148.716
C01778=1176.726,411.751,-85.687,-176.037,9.203,148.717
C01779=1176.722,411.998,-85.723,-176.037,9.205,148.717
C01780=1176.718,412.246,-85.760,-176.038,9.207,148.718
C01781=1176.715,412.493,-85.795,-176.037,9.209,148.718
C01782=1176.710,412.740,-85.832,-176.038,9.211,148.719
C01783=1176.706,412.987,-85.867,-176.038,9.213,148.720
C01784=1176.703,413.235,-85.903,-176.038,9.214,148.720
C01785=1176.699,413.482,-85.940,-176.038,9.217,148.721
C01786=1176.695,413.729,-85.975,-176.039,9.218,148.721
C01787=1176.690,413.977,-86.011,-176.039,9.220,148.722
C01788=1176.687,414.224,-86.048,-176.039,9.222,148.722
C01789=1176.683,414.472,-86.084,-176.039,9.224,148.723
C01790=1176.679,414.719,-86.120,-176.039,9.226,148.723
C01791=1176.675,414.967,-86.156,-176.039,9.228,148.724
C01792=1176.671,415.214,-86.192,-176.039,9.230,148.724
C01793=1176.667,415.457,-86.227,-176.040,9.232,148.725
C01794=1176.664,415.699,-86.263,-176.040,9.233,148.725
C01795=1176.662,415.941,-86.298,-176.040,9.235,148.726
C01796=1176.660,416.184,-86.333,-176.040,9.237,148.726
C01797=1176.660,416.427,-86.368,-176.040,9.238,148.727
C01798=1176.660,416.668,-86.403,-176.040,9.240,148.727
C01799=1176.662,416.910,-86.438,-176.040,9.242,148.728
C01800=1176.665,417.152,-86.473,-176.041,9.243,148.728
C01801=1176.244,417.154,-86.515,-176.044,9.254,148.732
C01802=1176.241,416.911,-86.481,-176.044,9.253,148.732
C01803=1176.239,416.666,-86.447,-176.043,9.251,148.731
C01804=1176.239,416.423,-86.411,-176.044,9.249,148.731
C01805=1176.239,416.179,-86.376,-176.043,9.248,148.730
C01806=1176.240,415.935,-86.340,-176.043,9.246,148.730
C01807=1176.242,415.691,-86.305,-176.043,9.244,148.729
C01808=1176.246,415.446,-86.270,-176.043,9.242,148.729
C01809=1176.250,415.203,-86.234,-176.042,9.241,148.728
C01810=1176.254,414.955,-86.197,-176.043,9.239,148.728
C01811=1176.258,414.708,-86.162,-176.042,9.237,148.727
C01812=1176.262,414.461,-86.125,-176.042,9.235,148.726
C01813=1176.266,414.213,-86.089,-176.042,9.233,148.726
C01814=1176.270,413.965,-86.053,-176.042,9.232,148.726
C01815=1176.273,413.718,-86.017,-176.041,9.229,148.725
C01816=1176.278,413.471,-85.981,-176.041,9.228,148.724
C01817=1176.281,413.224,-85.945,-176.041,9.225,148.724
C01818=1176.286,412.976,-85.908,-176.041,9.224,148.723
C01819=1176.289,412.728,-85.873,-176.041,9.221,148.723
C01820=1176.293,412.482,-85.837,-176.041,9.220,148.722
